    // M25 and M26 are coupled with M25 as the leader.
    // The motors cannot be set to always enabled, because they have brakes that
    // only activate when the motors are not moving. Due to the weight
    // of the frame, it appears that if the brake is not on, the motors
    // are moving constantly to keep the frame from falling. So essentially,
    // "is moving" is synonymous with "is enabled" for these motors which
    // results in the brake only applying if the motors are disabled. Setting M25
    // to only enable during motion, and M26 to NEVER means that
    // M25 will be enabled when commanded to move from EPICS but
    // for M26 the FB_MotionStage will not modify the bEnable boolean
    // in the state machine. Therefore, we can set the M26 bEnable
    // status based on the M25 bEnable status after the M25 FB_MotionStage
    // runs. But this also allows the brake to still activate when M26 is
    // not moving.
    Main.M25.nEnableMode := ENUM_StageEnableMode.NEVER ;
    // M26 bEnable is coupled to M25 bEnable below. Set M26 enable mode to NEVER
    // so that the function block does not try to set the bEnable bit unless
    // it detects an error. This allows the bEnable to be set outside of
    // the function block.
    Main.M26.nEnableMode := ENUM_StageEnableMode.NEVER ;

    Main.M27.nEnableMode := ENUM_StageEnableMode.DURING_MOTION ;
END_IF

stRenishawAbsEncMaster.Ref := 15370335;
stRenishawAbsEncSlave.Ref := 15347257;

// AutoCoupling
fbAutoCoupling(	nGantryTol 			:= 200000, // 50nm/count
                Master				:= Main.M25,
                MasterEnc			:= stRenishawAbsEncMaster,
                Slave				:= Main.M26,
                SlaveEnc			:= stRenishawAbsEncSlave,
                bExecuteCouple 		:= bExecuteCouple,
                bExecuteDecouple 	:= bExecuteDecouple,
);

// I don't think these 3 lines do anything but I am keeping for now.
// The FB_MotionStage overwrites the bAllEnable bit internally.
Main.M25.bAllEnable := Main.M25.bEnable AND GVL_EPS.bESTOP;
Main.M26.bAllEnable := Main.M26.bEnable AND GVL_EPS.bESTOP;
Main.M27.bAllEnable := Main.M27.bEnable AND GVL_EPS.bESTOP;

// Call Motion FB instance
IF NOT bDisableStateMachine THEN
    CASE nState OF
    -1:
        IF Main.M25.bExecute AND NOT (Main.M25.bError OR Main.M26.bError)  THEN
            Main.M25.bExecute := FALSE;
            Main.M25.bEnable := TRUE;
            nState := 0;
        ELSE
            Main.M25.bEnable := FALSE;
            Main.M25.bBrakeRelease := FALSE;
            Main.M26.bBrakeRelease := FALSE;
        END_IF
    0:
        tonDelay(IN:=TRUE, PT:=t#1s);
        IF tonDelay.Q THEN
            Main.M25.bBrakeRelease := TRUE;
            Main.M26.bBrakeRelease := TRUE;
            tonDelay(IN:=FALSE);
            nState := 1;
        ELSIF Main.M25.bError OR Main.M26.bError THEN
            nState := -1;
        END_IF
    1:
        tonDelay2(IN:=TRUE, PT:=t#1s);
        IF tonDelay2.Q THEN
            Main.M25.bExecute := TRUE;
            tonDelay2(IN:=FALSE);
            nState := 2;
        ELSIF Main.M25.bError OR Main.M26.bError THEN
            nState := -1;
        END_IF
    2:
        IF NOT Main.M25.bBusy AND NOT Main.M26.bBusy THEN
            nState := -1;
        END_IF
    100:
        nState := -1;
    END_CASE
END_IF

fbMotionYF1(stMotionStage:=Main.M25);

// Set the M26 bEnable equal to the M25 bEnable status to couple their enable bits together.
Main.M26.bEnable := Main.M25.bEnable;

fbMotionYF2(stMotionStage:=Main.M26);
fbMotionZF(stMotionStage:=Main.M27);

fbMeasureReferenceVelocity(
    stMotionStage:=Main.M25,
    nMicrostepsPerStep:=64,
    bBusy=>,
    fMeasuredReferenceVelocity=>
);

END_PROGRAM

// ---- Devices/FB_MeasureReferenceVelocity.TcPOU

FUNCTION_BLOCK FB_MeasureReferenceVelocity
VAR_IN_OUT
    stMotionStage: ST_MotionStage;
END_VAR
VAR_INPUT
    nMicrostepsPerStep: UINT := 64; // 64 for Beckhoff stepper drives EL7047, EL7037, EL7041, EL7031
END_VAR
VAR_OUTPUT
    bBusy: BOOL;
    fMeasuredReferenceVelocity: LREAL;
END_VAR
VAR
    nState: INT := -1;
    fbReadDriveAddress: MC_ReadDriveAddress;
    nMicrostepCounter AT %I*: UINT; // In microsteps (64 microsteps per step)
    bCounterOverflow AT %I*: BOOL;
    bCounterUnderflow AT %I*: BOOL;
    nMaxStepFrequencyBuffer: BYTE; // An enum corresponding to max step frequency
    fbReadCoEMaxStepFrequency: FB_ReadCoE;
    nMaxStepFrequency: UINT; // Fullsteps per Second
    fStartingInternalPosition: DINT;
    fEndingInternalPosition: DINT;
    fStartingEUPosition: LREAL;
    fEndingEUPosition: LREAL;
    fDeltaEUPosition: LREAL;
    fDeltaInternalPosition: LREAL;
    fDeltaSteps: LREAL;
    fEUPerStep: LREAL;

    rtOverflow: R_TRIG;
    rtUnderflow: R_TRIG;

    nDriveAddressReadState: INT := -1;
    bDriveAddressValid: BOOL;
END_VAR


CASE nDriveAddressReadState OF
-1:
    IF NOT bDriveAddressValid THEN
        nDriveAddressReadState := nDriveAddressReadState + 1;
        fbReadDriveAddress(
            Axis:=stMotionStage.Axis,
            Execute:=FALSE
        );
    END_IF
0: // Read drive address
    fbReadDriveAddress(
        Axis:=stMotionStage.Axis,
        Execute:=TRUE
    );
    IF NOT fbReadDriveAddress.Busy THEN
        nDriveAddressReadState := -1;
        bDriveAddressValid := TRUE;
    ELSIF fbReadDriveAddress.Error THEN
        nDriveAddressReadState := 100;
    END_IF
100:
    nDriveAddressReadState := -1;
END_CASE

CASE nState OF
-1:
    IF stMotionStage.bBusy AND bDriveAddressValid THEN
        nState := 0;
        fStartingInternalPosition := 0;
        fEndingInternalPosition := 0;
        rtOverflow(CLK:=bCounterOverflow);
        rtUnderflow(CLK:=bCounterUnderflow);
        fbReadCoEMaxStepFrequency(
            bExecute:=FALSE,
            pBuffer:=ADR(nMaxStepFrequencyBuffer)
        );
    ELSIF NOT bDriveAddressValid THEN
        nState := 100;
    END_IF
0: // A move has started so read the starting position information
    fbReadCoEMaxStepFrequency(
        bExecute:=TRUE,
        pBuffer:=ADR(nMaxStepFrequencyBuffer),
        sNetId:=stMotionStage.Axis.DriveAddress.NetID,
        nSlaveAddr:=stMotionStage.Axis.DriveAddress.SlaveAddress,
        nDesiredCoEIndex:=16#8012,
        nDesiredCoESubIndex:=5,
        nBufferLength:=1,
        bBusy=>,
        bError=>
    );
    IF fbReadCoEMaxStepFrequency.bBusy THEN
        nState := nState + 1;
    ELSIF fbReadCoEMaxStepFrequency.bError THEN
        nState := 100;
    END_IF
1:
    fbReadCoEMaxStepFrequency(
        bExecute:=TRUE,
        pBuffer:=ADR(nMaxStepFrequencyBuffer),
        sNetId:=stMotionStage.Axis.DriveAddress.NetID,
        nSlaveAddr:=stMotionStage.Axis.DriveAddress.SlaveAddress,
        nDesiredCoEIndex:=16#8012,
        nDesiredCoESubIndex:=5,
        nBufferLength:=1,
        bBusy=>,
        bError=>
    );
    IF NOT fbReadCoEMaxStepFrequency.bBusy THEN
        nState := nState + 1;
        fStartingEUPosition := stMotionStage.stAxisStatus.fActPosition;
        fStartingInternalPosition := nMicrostepCounter;

        CASE nMaxStepFrequencyBuffer OF
        0:
            nMaxStepFrequency := 1000;
        1:
            nMaxStepFrequency := 2000;
        2:
            nMaxStepFrequency := 4000;
        3:
            nMaxStepFrequency := 8000;
        4:
            nMaxStepFrequency := 16000;
        5:
            nMaxStepFrequency := 32000;
        END_CASE
    ELSIF fbReadCoEMaxStepFrequency.bError THEN
        nState := 100;
    END_IF
2: // Wait until the move ends and then read the last position information
    rtOverflow(CLK:=bCounterOverflow);
    rtUnderflow(CLK:=bCounterUnderflow);
    IF rtOverflow.Q THEN
        fEndingInternalPosition := fEndingInternalPosition + 65535;
    ELSIF rtUnderflow.Q THEN
        fEndingInternalPosition := fEndingInternalPosition - 65535;
    END_IF
    IF NOT stMotionStage.bBusy THEN
        nState := nState + 1;
        fEndingEUPosition := stMotionStage.stAxisStatus.fActPosition;
        fEndingInternalPosition := fEndingInternalPosition + nMicrostepCounter;
    END_IF
3: // Calculate the reference velocity from the measured move
    fDeltaEUPosition := fEndingEUPosition - fStartingEUPosition;
    fDeltaInternalPosition := fEndingInternalPosition - fStartingInternalPosition;
    fDeltaSteps := fDeltaInternalPosition / UINT_TO_LREAL(nMicrostepsPerStep);

    IF fDeltaSteps <> 0 THEN
        fEUPerStep := fDeltaEUPosition / fDeltaSteps;

        fMeasuredReferenceVelocity := UINT_TO_LREAL(nMaxStepFrequency) * fEUPerStep;
        nState := -1;
    ELSE
        nState := 100;
        fMeasuredReferenceVelocity := 0;
    END_IF
100: // Reserve for error handling
    nState := -1;
END_CASE

END_FUNCTION_BLOCK

// ---- Devices/FB_ReadCoE.TcPOU

FUNCTION_BLOCK FB_ReadCoE
VAR_INPUT
    bExecute: BOOL;
    pBuffer: PVOID; // ADR(buffer)
    sNetId: T_AmsNetId; // Have to be entered
    nSlaveAddr: UINT; // Have to be entered
    nDesiredCoEIndex: WORD; // Ex: CoE 16#9000 (9000:1)
    nDesiredCoESubIndex: Byte; // Ex: CoE 1 (9000:1)
    nBufferLength: UDINT; // number of bytes in the CoE to be read
END_VAR
VAR_OUTPUT
    bBusy: BOOL;
    bError: BOOL;
END_VAR
VAR
    fbCoERead: FB_EcCoESdoRead; // Function Block for reading from CoE
    nState: INT := -1; // RW-status
    rtExecute: R_TRIG;
END_VAR


CASE nState OF
-1:
    rtExecute(CLK:=bExecute);
    IF rtExecute.Q THEN
        nState := 0;
        bBusy := TRUE;
        bError := FALSE;
    ELSE
        bBusy := FALSE;
    END_IF
0:
   // Read entry
    fbCoERead(
       sNetId:= sNetId,
       nSlaveAddr:= nSlaveAddr,
       nSubIndex:= nDesiredCoeSubIndex,
       nIndex:= nDesiredCoEIndex,
       pDstBuf:= pBuffer,
       cbBufLen:= nBufferLength,
       bExecute:= FALSE,
       tTimeout:= T#1S
   );
   fbCoERead(
       sNetId:= sNetId,
       nSlaveAddr:= nSlaveAddr,
       nSubIndex:= nDesiredCoeSubIndex,
       nIndex:= nDesiredCoEIndex,
       pDstBuf:= pBuffer,
       cbBufLen:= nBufferLength,
       bExecute:= TRUE,
       tTimeout:= T#1S
   );
   nState := nState + 1; // Next state
1: // Execute CoE read until done
    fbCoERead(
       sNetId:= sNetId,
       nSlaveAddr:= nSlaveAddr,
       nSubIndex:= nDesiredCoeSubIndex,
       nIndex:= nDesiredCoEIndex,
       pDstBuf:= pBuffer,
       cbBufLen:= nBufferLength,
       bExecute:= TRUE,
       tTimeout:= T#1S
    );
    IF fbCoERead.bError THEN
      nState := 100;     // Error case
    ELSE
        IF NOT fbCoERead.bBusy THEN
            nState := -1;    // Done
            bBusy := FALSE;
        END_IF
    END_IF
100: // Error handling..
    nState := -1;
    bBusy := FALSE;
    bError := TRUE;
END_CASE

END_FUNCTION_BLOCK

// ---- Spectometer Arm POUs/PRG_DET_CHAMBER.TcPOU

PROGRAM PRG_DET_CHAMBER
VAR
    bInit: BOOL := TRUE;
    fbMotionXDC: FB_MotionStage;
    fbMotionRyDC: FB_MotionStage;
    fbMotionZDC: FB_MotionStage;
END_VAR


// Det. Chmber
IF bInit THEN
    bInit :=FALSE;
    Main.M22.bHardwareEnable:= TRUE;
    Main.M22.bPowerSelf:= TRUE;
    Main.M22.nBrakeMode:= ENUM_StageBrakeMode.NO_BRAKE;
    Main.M22.nEnableMode := ENUM_StageEnableMode.DURING_MOTION ;
    Main.M22.fVelocity := 0.1;

    Main.M23.bHardwareEnable:= TRUE;
    Main.M23.bPowerSelf:= TRUE;
    Main.M23.nBrakeMode:= ENUM_StageBrakeMode.NO_BRAKE;
    Main.M23.nEnableMode := ENUM_StageEnableMode.DURING_MOTION ;
    Main.M23.fVelocity := 0.1;

    Main.M24.bHardwareEnable:= TRUE;
    Main.M24.bPowerSelf:= TRUE;
    Main.M24.nBrakeMode:= ENUM_StageBrakeMode.NO_BRAKE;
    Main.M24.nEnableMode := ENUM_StageEnableMode.ALWAYS ; // This axis should always be enables due to belows
    Main.M24.fVelocity := 0.1;
END_IF;


fbMotionXDC(stMotionStage:= Main.M22);
fbMotionRyDC(stMotionStage:= Main.M23);
fbMotionZDC(stMotionStage:= Main.M24);

END_PROGRAM

// ---- Spectometer Arm POUs/PRG_DET_SLIT.TcPOU

PROGRAM PRG_DET_SLIT
VAR
    {attribute 'pytmc' := 'pv: QRIX:DETSL'}
    fbSlits_Det: FB_Slits;
    bExecuteMotion: BOOL := TRUE;
    bMoveOk: BOOL :=TRUE;
    bInit:BOOL:=TRUE;
END_VAR


// 4 jaws slit

IF bInit THEN
    bInit := FALSE;

    Main.M18.nBrakeMode := ENUM_StageBrakeMode.NO_BRAKE;
    Main.M18.bHardwareEnable := TRUE;
    Main.M18.bPowerSelf := TRUE;
    Main.M18.fVelocity := 0.1;

    Main.M19.nBrakeMode := ENUM_StageBrakeMode.NO_BRAKE;
    Main.M19.bHardwareEnable := TRUE;
    Main.M19.bPowerSelf := TRUE;
    Main.M19.fVelocity := 0.1;

    Main.M20.nBrakeMode := ENUM_StageBrakeMode.NO_BRAKE;
    Main.M20.bHardwareEnable := TRUE;
    Main.M20.bPowerSelf := TRUE;
    Main.M20.fVelocity := 0.1;

    Main.M21.nBrakeMode := ENUM_StageBrakeMode.NO_BRAKE;
    Main.M21.bHardwareEnable := TRUE;
    Main.M21.bPowerSelf := TRUE;
    Main.M21.fVelocity := 0.1;

    Main.M18.nEnableMode := ENUM_StageEnableMode.DURING_MOTION ;
    Main.M19.nEnableMode := ENUM_StageEnableMode.DURING_MOTION ;
    Main.M20.nEnableMode := ENUM_StageEnableMode.DURING_MOTION ;
    Main.M21.nEnableMode := ENUM_StageEnableMode.DURING_MOTION ;
END_IF
fbSlits_Det(	i_DevName:=					'DET_SLITS',
                stTopBlade:=				Main.M20,
                stBottomBlade:=				Main.M21,
                stLeftBlade:=				Main.M18,
                stRightBlade:=				Main.M19,
                io_fbFFHWO:=				GVL_PMPS.fbFastFaultOutput1,
                fbArbiter:=					GVL_PMPS.fbArbiter,
                bExecuteMotion:=			bExecuteMotion,
                bMoveOk:=					bMoveOk
);

END_PROGRAM

// ---- Devices/FB_Slits.TcPOU

FUNCTION_BLOCK FB_Slits
VAR_IN_OUT
    stTopBlade: ST_MotionStage;
    stBottomBlade: ST_MotionStage;
    stLeftBlade: ST_MotionStage; // Left Slit from upstream view
    stRightBlade: ST_MotionStage; // Right Slit from upstream view
    bExecuteMotion:BOOL ;
    io_fbFFHWO    :    FB_HardwareFFOutput;
    fbArbiter: FB_Arbiter();
END_VAR

VAR_INPUT

    {attribute 'pytmc' := '
    pv: PMPS_OK;
    io: i;
    field: ZNAM False
    field: ONAM True
    '}
    bMoveOk:BOOL;

    (*Offsets*)
    {attribute 'pytmc' := '
    pv: Offset_Top;
    io: io;
    '}
    rEncoderOffsetTop: REAL;
    {attribute 'pytmc' := '
    pv: ZeroOffset_Bottom;
    io: io;
    '}
    rEncoderOffsetBottom: REAL;

    {attribute 'pytmc' := 'pv: ZeroOffset_Left; io: io;'}
    rEncoderOffsetLeft: REAL;

    {attribute 'pytmc' := '
    pv: ZeroOffset_Right;
    io: io;
    '}
    rEncoderOffsetRight: REAL;
    i_DevName : STRING; //device name for FFO and PMPS diagnostics
    {attribute 'pytmc' := '
    pv: Home;
    io: i;
    field: ZNAM False
    field: ONAM True
    '}
    bHome:BOOL:=FALSE;
END_VAR

VAR
    fbTopBlade: FB_MotionStage;
    fbBottomBlade: FB_MotionStage;
    fbLeftBlade: FB_MotionStage;
    fbRightBlade: FB_MotionStage;
    fPosTopBlade: LREAL;
    fPosBottomBlade: LREAL;
    fPosLeftBlade: LREAL;
    fPosRightBlade: LREAL;

    bCollisionLimitationVert: BOOL;
    bCollisionLimitationHorz: BOOL;

    (*Motion Parameters*)
    fSmallDelta: LREAL := 0.01;
    fBigDelta: LREAL := 20;
    fMaxVelocity: LREAL := 0.5;
    fHighAccel: LREAL := 0.8;
    fLowAccel: LREAL := 0.1;

    stTop: ST_PositionState;
    stBOTTOM: ST_PositionState;
    stLeft: ST_PositionState;
    stRight: ST_PositionState;

    {attribute 'pytmc' := 'pv: TOP'}
    fbTop: FB_StatePTPMove;
    {attribute 'pytmc' := 'pv: BOTTOM'}
    fbBottom: FB_StatePTPMove;
    {attribute 'pytmc' := 'pv: LEFT'}
    fbLeft: FB_StatePTPMove;
    {attribute 'pytmc' := 'pv: RIGHT'}
    fbRight: FB_StatePTPMove;

    (*EPICS pvs*)
    {attribute 'pytmc' := '
    pv: XWID_REQ;
    io: io;
    '}
    rReqApertureSizeX : REAL;
    {attribute 'pytmc' := '
    pv: YWID_REQ;
    io: io;
    '}
    rReqApertureSizeY : REAL;
    {attribute 'pytmc' := '
    pv: XCEN_REQ;
    io: io;
    '}
    rReqCenterX: REAL;
    {attribute 'pytmc' := '
    pv: YCEN_REQ;
    io: io;
    '}
    rReqCenterY: REAL;

    {attribute 'pytmc' := '
    pv: ACTUAL_XWIDTH;
    io: io;
    '}
    rActApertureSizeX : REAL;

    {attribute 'pytmc' := '
    pv: ACTUAL_YWIDTH;
    io: io;
    '}
    rActApertureSizeY : REAL;
    {attribute 'pytmc' := '
    pv: ACTUAL_XCENTER;
    io: io;
    '}
    rActCenterX: REAL;
    {attribute 'pytmc' := '
    pv: ACTUAL_YCENTER;
    io: io;
    '}
    rActCenterY: REAL;

    {attribute 'pytmc' := '
    pv: XCEN_SETZERO;
    io: io;
    '}
    rSetCenterX: BOOL;
    {attribute 'pytmc' := '
    pv: YCEN_SETZERO;
    io: io;
    '}
    rSetCenterY: BOOL;


    {attribute 'pytmc' := '
    pv: OPEN;
    io: io;
    field: ZNAM False
    field: ONAM True
    '}
    bOpen: BOOL;

    {attribute 'pytmc' := '
    pv: CLOSE;
    io: io;
    field: ZNAM False
    field: ONAM True
    '}
    bClose: BOOL;

    {attribute 'pytmc' := '
    pv: BLOCK;
    io: io;
    field: ZNAM False
    field: ONAM True
    '}
    bBlock: BOOL;


     {attribute 'pytmc' := '
    pv: HOME_READY;
    io: i;
    field: ZNAM False
    field: ONAM True
    '}
    bHomeReady:BOOL:=FALSE;


    //Local variables
    bInit: BOOL :=true;
    rTrig_Block: R_TRIG;
    rTrig_Open: R_TRIG;
    rTrig_Close: R_TRIG;

    //old values
    rOldReqApertureSizeX : REAL;
    rOldReqApertureSizeY : REAL;
    rOldReqCenterX: REAL;
    rOldReqCenterY: REAL;

    bExecuteMotionX: BOOL;
    bExecuteMotionY: BOOL;


    fPosBlock: LREAL;
    fPosClose: LREAL;
    fPosOpen: LREAL;

    stSetPositionOptions:ST_SetPositionOptions;
    fbSetPosition_TOP: MC_SetPosition;
    fbSetPosition_Bottom: MC_SetPosition;
    fbSetPosition_Left: MC_SetPosition;
    fbSetPosition_Right: MC_SetPosition;

    // For logging
    fbLogger : FB_LogMessage := (eSubsystem:=E_SubSystem.MOTION);
    tErrorPresent : R_TRIG;
    tAction : R_TRIG;
    tOverrideActivated : R_TRIG;

    FFO    :    FB_FastFault :=(
        i_DevName := 'Slits',
        i_Desc := 'Fault occurs when center is greated than that requested',
        i_TypeCode := 16#1010);


    bTest: BOOL;

    AptArrayStatus AT %Q* : ST_PMPS_Aperture_IO;
    AptArrayReq AT %I* : ST_PMPS_Aperture_IO;

    fbPower: MC_Power;
END_VAR


// Initialize
ACT_init();
// Instantiate Function block for all the blades
ACT_Motion();
//SET and GET the requested and Actual values
ACT_CalculatePositions();

// Software Limits to protect blades
ACT_VirtualLimitSW();

ACTION ACT_BLOCK:

rTrig_Block (CLK:= bBlock);
rTrig_Open (CLK:= bOpen);
rTrig_Close (CLK:= bClose);

if (rTrig_Block.Q) THEN
    //BLOCK

    bBlock := false;
END_IF

if (rTrig_Open.Q) THEN


    bOpen := false;
END_IF

if (rTrig_Close.Q) THEN


    bClose := false;
END_IF
END_ACTION

ACTION ACT_CalculatePositions:

//check if requested center or gap has changed
//check that the requested values are within acceptable motion range
IF (rOldReqApertureSizeX <> rReqApertureSizeX) THEN
        rOldReqApertureSizeX := rReqApertureSizeX;
        bExecuteMotionX := TRUE;
        fbLogger(sMsg:='Requested new X gap.', eSevr:=TcEventSeverity.Verbose);
END_IF

IF (rOldReqCenterX <> rReqCenterX) THEN
    rOldReqCenterX := rReqCenterX;
    bExecuteMotionX := TRUE;
    fbLogger(sMsg:='Requested new X center', eSevr:=TcEventSeverity.Verbose);
   // ELSE
      //  rReqCenterX := rActCenterX;
END_IF

IF (rOldReqApertureSizeY <> rReqApertureSizeY) THEN
        rOldReqApertureSizeY := rReqApertureSizeY;
        bExecuteMotionY := TRUE;
        fbLogger(sMsg:='Requested new Y gap.', eSevr:=TcEventSeverity.Verbose);

END_IF

IF (rOldReqCenterY <> rReqCenterY) THEN
    rOldReqCenterY := rReqCenterY;
    bExecuteMotionY := TRUE;
    fbLogger(sMsg:='Requested new Y center.', eSevr:=TcEventSeverity.Verbose);
   // ELSE
      //  rReqCenterY := rActCenterY;
END_IF


//Calculate requested target positions from requested gap and center
fPosTopBlade := (rReqApertureSizeY/2) + (rReqCenterY + rEncoderOffsetTop) ;
fPosBottomBlade := (-1*rReqApertureSizeY/2) + (rReqCenterY+rEncoderOffsetBottom);

fPosLeftBlade := (rReqApertureSizeX/2) + (rReqCenterX + rEncoderOffsetLeft);
fPosRightBlade := (-1*rReqApertureSizeX/2) + (rReqCenterX + rEncoderOffsetRight);


//Calculate actual gap and center from actual stages positions
rActApertureSizeX := LREAL_TO_REAL((stLeftBlade.stAxisStatus.fActPosition - rEncoderOffsetLeft) - (stRightBlade.stAxisStatus.fActPosition- rEncoderOffsetRight));

rActApertureSizeY := LREAL_TO_REAL((stTopBlade.stAxisStatus.fActPosition - rEncoderOffsetTop) - (stBottomBlade.stAxisStatus.fActPosition - rEncoderOffsetBottom));

rActCenterX := LREAL_TO_REAL((((stLeftBlade.stAxisStatus.fActPosition - rEncoderOffsetLeft)  + (stRightBlade.stAxisStatus.fActPosition - rEncoderOffsetRight ))/2));

rActCenterY := LREAL_TO_REAL((((stTopBlade.stAxisStatus.fActPosition - rEncoderOffsetTop) + (stBottomBlade.stAxisStatus.fActPosition - rEncoderOffsetBottom))/2));


// Prevent collision
bCollisionLimitationHorz	:= (rActApertureSizeX > -0.1);
bCollisionLimitationVert	:= (rActApertureSizeY > -0.1);
END_ACTION

ACTION ACT_Init:

//  init the motion stages parameters
IF ( bInit) THEN
    stTopBlade.bHardwareEnable := TRUE;
    stBottomBlade.bHardwareEnable := TRUE;
    stLeftBlade.bHardwareEnable := TRUE;
    stRightBlade.bHardwareEnable := TRUE;
    stTopBlade.bPowerSelf :=FALSE;
    stBottomBlade.bPowerSelf :=FALSE;
    stLeftBlade.bPowerSelf :=FALSE;
    stRightBlade.bPowerSelf :=FALSE;
    stTopBlade.nBrakeMode := ENUM_StageBrakeMode.NO_BRAKE;
    stBottomBlade.nBrakeMode := ENUM_StageBrakeMode.NO_BRAKE;
    stLeftBlade.nBrakeMode := ENUM_StageBrakeMode.NO_BRAKE;
    stRightBlade.nBrakeMode := ENUM_StageBrakeMode.NO_BRAKE;
    FFO.i_DevName := i_DevName;
END_IF
END_ACTION

ACTION ACT_Motion:

// Instantiate Function block for all the blades
fbTopBlade(stMotionStage:=stTopBlade);
fbBottomBlade(stMotionStage:=stBottomBlade);
fbLeftBlade(stMotionStage:=stLeftBlade);
fbRightBlade(stMotionStage:=stRightBlade);



// PTP Motion for each blade
stTop.sName := 'Top';
stTop.fPosition := fPosTopBlade;
stTop.fDelta := fSmallDelta;
stTop.fVelocity := fMaxVelocity;
stTop.fAccel := fHighAccel;
stTop.fDecel := fHighAccel;

stBOTTOM.sName := 'Bottom';
stBOTTOM.fPosition := fPosBottomBlade;
stBOTTOM.fDelta := fSmallDelta;
stBOTTOM.fVelocity := fMaxVelocity;
stBOTTOM.fAccel := fHighAccel;
stBOTTOM.fDecel := fHighAccel;

stLeft.sName := 'Left';
stLeft.fPosition := fPosLeftBlade;
stLeft.fDelta := fSmallDelta;
stLeft.fVelocity := fMaxVelocity;
stLeft.fAccel := fHighAccel;
stLeft.fDecel := fHighAccel;

stRight.sName := 'Right';
stRight.fPosition := fPosRightBlade;
stRight.fDelta := fSmallDelta;
stRight.fVelocity := fMaxVelocity;
stRight.fAccel := fHighAccel;
stRight.fDecel := fHighAccel;

IF (bExecuteMotionY) THEN
    fbTop.bExecute := fbBottom.bExecute := bExecuteMotionY;
    bExecuteMotionY:= FALSE;
END_IF

IF (bExecuteMotionX) THEN
    fbLeft.bExecute := fbRight.bExecute := bExecuteMotionX;
    bExecuteMotionX:= FALSE;
END_IF


fbTop(
    stPositionState:=stTop,
    bMoveOk:=bMoveOk,
    stMotionStage:=stTopBlade);

fbBottom(
    stPositionState:=stBOTTOM,
    bMoveOk:=bMoveOk,
    stMotionStage:=stBottomBlade);

fbLeft(
    stPositionState:=stLeft,
    bMoveOk:=bMoveOk,
    stMotionStage:=stLeftBlade);

fbRight(
    stPositionState:=stRight,
    bMoveOk:=bMoveOk,
    stMotionStage:=stRightBlade);
END_ACTION

ACTION ACT_VirtualLimitSW:

// Force set to false
stLeftBlade.bPowerSelf := stRightBlade.bPowerSelf := stTopBlade.bPowerSelf := stBottomBlade.bPowerSelf := FALSE;

// Set SafetyReady flags manually
stTopBlade.bSafetyReady:= TRUE;
stBottomBlade.bSafetyReady:= TRUE;
stLeftBlade.bSafetyReady:= TRUE;
stRightBlade.bSafetyReady:= TRUE;


// Note: FB_MotionStage calls FB_SetEnables internally that overwrites .bAllForwardEnable/.bAllBackwardEnable flags

fbPower(
    Axis := stTopBlade.Axis,
    Enable := stTopBlade.bAllEnable,
    Enable_Positive := stTopBlade.bAllForwardEnable,
    Enable_Negative := stTopBlade.bAllBackwardEnable AND bCollisionLimitationVert,
    Override := 100.000
);
fbPower(
    Axis := stBottomBlade.Axis,
    Enable := stBottomBlade.bAllEnable,
    Enable_Positive := stBottomBlade.bAllForwardEnable AND bCollisionLimitationVert,
    Enable_Negative := stBottomBlade.bAllBackwardEnable,
    Override := 100.000
);
fbPower(
    Axis := stLeftBlade.Axis,
    Enable := stLeftBlade.bAllEnable,
    Enable_Positive := stLeftBlade.bAllForwardEnable,
    Enable_Negative := stLeftBlade.bAllBackwardEnable AND bCollisionLimitationHorz,
    Override := 100.000
);
fbPower(
    Axis := stRightBlade.Axis,
    Enable := stRightBlade.bAllEnable,
    Enable_Positive := stRightBlade.bAllForwardEnable AND bCollisionLimitationHorz,
    Enable_Negative := stRightBlade.bAllBackwardEnable,
    Override := 100.000
);
END_ACTION

END_FUNCTION_BLOCK

// ---- Spectometer Arm POUs/PRG_DET_FRAME.TcPOU

PROGRAM PRG_DET_FRAME
VAR
    bInit: BOOL := TRUE;
    {attribute 'pytmc' := '
        pv: QRIX:SA:bError
        io: i
    '}
    bError: BOOL := FALSE;
    {attribute 'pytmc' := '
        pv: QRIX:SA:bBusy
        io: i
    '}
    bBusy: BOOL;
    {attribute 'pytmc' := '
        pv: QRIX:SA:bMotorsBusy
        io: i
    '}
    bMotorsBusy: BOOL;
    {attribute 'pytmc' := 'pv: QRIX:SA:bResetError'}
    bResetError: BOOL := FALSE;
    {attribute 'pytmc' := 'pv: QRIX:SA:EnableJackOff'}
    bEnableJackOff: BOOL;
    {attribute 'pytmc' := 'pv: QRIX:SA:EnableLevitation'}
    bEnableLevitation: BOOL;
    {attribute 'pytmc' := 'pv: QRIX:SA:EnableLanding'}
    bEnableLanding: BOOL;
    {attribute 'pytmc' := 'pv: QRIX:DF:EnableAdjustingRoll'}
    bEnableAdjustingRoll: BOOL;
    {attribute 'pytmc' := 'pv: QRIX:DF:EnableAdjustingPitch'}
    bEnableAdjustingPitch: BOOL;
    {attribute 'pytmc' := 'pv: QRIX:DF:EnableAdjustingHeight'}
    bEnableAdjustingHeight: BOOL;

    tonWaitToStabilize: TON;

    tonSV2Open: TON;
    tonSV1Close: TON;

    tonDelayTrig: TON;

    iStepJackOff: INT := 1;
    iStepAdjustingRoll : INT := 1;
    iStepAdjustingPitch : INT := 1;
    iStepAdjustingHeight : INT := 1;

    trigDone: F_TRIG;

    fDistanceX: LREAL := 2.114; // in m
    fDistanceZ: LREAL := 2.142; // in m

    fPositionThreshold: LREAL := 0.02; // mm
    fPositionMaxDeviation: LREAL := 10.0; // mm
    fPitchThreshold: LREAL := 0.02; // mrad
    fRollThreshold: LREAL := 0.02; // mrad

    {attribute 'pytmc' := '
        pv: QRIX:SA:fRollTarget
        io: io
    '}
    fRollTarget : LREAL;

    {attribute 'pytmc' := 'pv: QRIX:F'}
    fbYDFMotion: FB_3AxesJack;

    fbReset_M15: MC_RESET;
    fbReset_M16: MC_RESET;
    fbReset_M17: MC_RESET;

    nActiveSequenceIterationCount: UINT := 1;
    nSequenceIterationCount: UINT := 3;

    // EPS settings to prevent jacks from moving too far out of range of each other.
    EPS_YDF1_Up   : FB_EPS;
    EPS_YDF1_Down : FB_EPS;
    EPS_YDF2_Up   : FB_EPS;
    EPS_YDF2_Down : FB_EPS;
    EPS_YDF3_Up   : FB_EPS;
    EPS_YDF3_Down : FB_EPS;

    {attribute 'pytmc' := '
        pv: QRIX:SA:rJackingSpeed
        io: io
    '}
    rJackingSpeed: LREAL := 0.05;
    {attribute 'pytmc' := '
        pv: QRIX:SA:rJackingAccel
        io: io
    '}
    rJackingAccel: LREAL := 0.005;

    {attribute 'pytmc' := '
        pv: QRIX:SA:bStopAxes
        io: io
    '}
    bStopAxes: BOOL;

    {attribute 'TcLinkTo' := 'TIIB[Rack#2D LinearGaugeAmp (SC-HG1-ETC)]^Process Data(In)  TxPDO-Map^Sensor Warning}
    bLinearGaugeWarning AT %I* : BOOL;
    {attribute 'TcLinkTo' := 'TIIB[Rack#2D LinearGaugeAmp (SC-HG1-ETC)]^Process Data(In)  TxPDO-Map^Sensor Error}
    bLinearGaugeError AT %I* : BOOL;

    {attribute 'TcLinkToOSO' := '<0,1,2>TINC^NC-Task 1 SAF^Axes^M15 - YDF1^Enc^Inputs^In^nState1'}
    bLinearGaugeYDF1Ready AT %Q* : BOOL;
    {attribute 'TcLinkToOSO' := '<0,1,2>TINC^NC-Task 1 SAF^Axes^M16 - YDF2^Enc^Inputs^In^nState1'}
    bLinearGaugeYDF2Ready AT %Q* : BOOL;
    {attribute 'TcLinkToOSO' := '<0,1,2>TINC^NC-Task 1 SAF^Axes^M17 - YDF3^Enc^Inputs^In^nState1'}
    bLinearGaugeYDF3Ready AT %Q* : BOOL;
END_VAR


IF bInit THEN
    bInit := FALSE;

    Main.M15.nBrakeMode := ENUM_StageBrakeMode.NO_BRAKE;
    Main.M15.bHardwareEnable := TRUE;
    Main.M15.bPowerSelf := TRUE;

    Main.M16.nBrakeMode := ENUM_StageBrakeMode.NO_BRAKE;
    Main.M16.bHardwareEnable := TRUE;
    Main.M16.bPowerSelf := TRUE;

    Main.M17.nBrakeMode := ENUM_StageBrakeMode.NO_BRAKE;
    Main.M17.bHardwareEnable := TRUE;
    Main.M17.bPowerSelf := TRUE;

    Main.M15.nEnableMode := ENUM_StageEnableMode.DURING_MOTION;
    Main.M16.nEnableMode := ENUM_StageEnableMode.DURING_MOTION;
    Main.M17.nEnableMode := ENUM_StageEnableMode.DURING_MOTION;
END_IF;

// FRAME JACKS EPS RESTRICTIONS
// YDF1 Disable movement in upward (positive/forward) direction.
EPS_YDF1_Up(eps:=Main.M15.stEPSForwardEnable);
EPS_YDF1_Up.setDescription('UPWARD MOVEMENT ALLOWED IF: YDF1 - YDF2 < 10mm AND YDF1 - YDF3 < 10mm |'); // SET DESCRIPTION FOR BYTE INDICATOR LABELS
// Prevent YDF1 from rising any more if it is more than fPositionMaxDeviation above YDF2
EPS_YDF1_Up.setBit(nBits:= 1, bValue:= Main.M15.stAxisStatus.fActPosition - Main.M16.stAxisStatus.fActPosition < fPositionMaxDeviation);
// Prevent YDF1 from rising any more if it is more than fPositionMaxDeviation above YDF3
EPS_YDF1_Up.setBit(nBits:= 0, bValue:= Main.M15.stAxisStatus.fActPosition - Main.M17.stAxisStatus.fActPosition < fPositionMaxDeviation);

// YDF1 Disable movement in downward (negative/downward) direction.
EPS_YDF1_Down(eps:=Main.M15.stEPSBackwardEnable);
EPS_YDF1_Down.setDescription('DOWNWARD MOVEMENT ALLOWED IF: YDF1 - YDF2 > -10mm AND YDF1 - YDF3 > -10mm |'); // SET DESCRIPTION FOR BYTE INDICATOR LABELS
// Prevent YDF1 from lowering any more if it is more than fPositionMaxDeviation below YDF2
EPS_YDF1_Down.setBit(nBits:= 1, bValue:= Main.M15.stAxisStatus.fActPosition - Main.M16.stAxisStatus.fActPosition > -fPositionMaxDeviation);
// Prevent YDF1 from lowering any more if it is more than fPositionMaxDeviation below YDF3
EPS_YDF1_Down.setBit(nBits:= 0, bValue:= Main.M15.stAxisStatus.fActPosition - Main.M17.stAxisStatus.fActPosition > -fPositionMaxDeviation);

// YDF2 Disable movement in upward (positive/forward) direction.
EPS_YDF2_Up(eps:=Main.M16.stEPSForwardEnable);
EPS_YDF2_Up.setDescription('UPWARD MOVEMENT ALLOWED IF:  YDF2 - YDF1 < 10mm AND YDF2 - YDF3 < 10mm |'); // SET DESCRIPTION FOR BYTE INDICATOR LABELS
// Prevent YDF2 from rising any more if it is more than fPositionMaxDeviation above YDF1
EPS_YDF2_Up.setBit(nBits:= 1, bValue:= Main.M16.stAxisStatus.fActPosition - Main.M15.stAxisStatus.fActPosition < fPositionMaxDeviation);
// Prevent YDF2 from rising any more if it is more than fPositionMaxDeviation above YDF3
EPS_YDF2_Up.setBit(nBits:= 0, bValue:= Main.M16.stAxisStatus.fActPosition - Main.M17.stAxisStatus.fActPosition < fPositionMaxDeviation);

// YDF2 Disable movement in downward (negative/downward) direction.
EPS_YDF2_Down(eps:=Main.M16.stEPSBackwardEnable);
EPS_YDF2_Down.setDescription('DOWNWARD MOVEMENT ALLOWED IF: YDF2 - YDF1 > -10mm AND YDF2 - YDF3 > -10mm |'); // SET DESCRIPTION FOR BYTE INDICATOR LABELS
// Prevent YDF2 from lowering any more if it is more than fPositionMaxDeviation below YDF1
EPS_YDF2_Down.setBit(nBits:= 1, bValue:= Main.M16.stAxisStatus.fActPosition - Main.M15.stAxisStatus.fActPosition > -fPositionMaxDeviation);
// Prevent YDF2 from lowering any more if it is more than fPositionMaxDeviation below YDF3
EPS_YDF2_Down.setBit(nBits:= 0, bValue:= Main.M16.stAxisStatus.fActPosition - Main.M17.stAxisStatus.fActPosition > -fPositionMaxDeviation);

// YDF3 Disable movement in upward (positive/forward) direction.
EPS_YDF3_Up(eps:=Main.M17.stEPSForwardEnable);
EPS_YDF3_Up.setDescription('UPWARD MOVEMENT ALLOWED IF: YDF3 - YDF2 < 10mm AND YDF3 - YDF1 < 10mm |'); // SET DESCRIPTION FOR BYTE INDICATOR LABELS
// Prevent YDF3 from rising any more if it is more than fPositionMaxDeviation above YDF2
EPS_YDF3_Up.setBit(nBits:= 1, bValue:= Main.M17.stAxisStatus.fActPosition - Main.M16.stAxisStatus.fActPosition < fPositionMaxDeviation);
// Prevent YDF3 from rising any more if it is more than fPositionMaxDeviation above YDF1
EPS_YDF3_Up.setBit(nBits:= 0, bValue:= Main.M17.stAxisStatus.fActPosition - Main.M15.stAxisStatus.fActPosition < fPositionMaxDeviation);

// YDF3 Disable movement in downward (negative/downward) direction.
EPS_YDF3_Down(eps:=Main.M17.stEPSBackwardEnable);
EPS_YDF3_Down.setDescription('DOWNWARD MOVEMENT ALLOWED IF: YDF3 - YDF2 > -10mm AND YDF3 - YDF1 > -10mm |'); // SET DESCRIPTION FOR BYTE INDICATOR LABELS
// Prevent YDF3 from lowering any more if it is more than fPositionMaxDeviation below YDF2
EPS_YDF3_Down.setBit(nBits:= 1, bValue:= Main.M17.stAxisStatus.fActPosition - Main.M16.stAxisStatus.fActPosition > -fPositionMaxDeviation);
// Prevent YDF3 from lowering any more if it is more than fPositionMaxDeviation below YDF1
EPS_YDF3_Down.setBit(nBits:= 0, bValue:= Main.M17.stAxisStatus.fActPosition - Main.M15.stAxisStatus.fActPosition > -fPositionMaxDeviation);

GVL_Sensor.bFloating := GVL_Sensor.stPS1.fValue > 0.3 AND GVL_Sensor.stPS2.fValue > 0.18 AND GVL_Sensor.stPS3.fValue > 0.15;

bMotorsBusy := Main.M15.bBusy OR Main.M16.bBusy OR Main.M17.bBusy;

IF Main.M15.bError OR Main.M16.bError OR Main.M17.bError THEN
    bError := TRUE;
    iStepJackOff := -1;
    iStepAdjustingRoll := -1;
    iStepAdjustingPitch := -1;
    iStepAdjustingHeight := -1;
    IF NOT Main.M15.bError THEN
        Main.M15.bReset := TRUE;
    END_IF;
    IF NOT Main.M16.bError THEN
        Main.M16.bReset := TRUE;
    END_IF;
    IF NOT Main.M17.bError THEN
        Main.M17.bReset := TRUE;
    END_IF;
END_IF

ACT_1_JACK_OFF();
ACT_2_Levitation();
ACT_3_Landing();
ACT_4_AdjustingRoll();
ACT_5_AdjustingPitch();
ACT_6_AdjustingHeight();
ACT_ResetError();

bLinearGaugeYDF1Ready := NOT bLinearGaugeError;
bLinearGaugeYDF2Ready := NOT bLinearGaugeError;
bLinearGaugeYDF3Ready := NOT bLinearGaugeError;

fbYDFMotion(
    bMoveOk			  := GVL_EPS.bESTOP,
    stJack1Axis		  := Main.M16,
    stJack2Axis		  := Main.M15,
    stJack3Axis		  := Main.M17,
    rDistanceX        := fDistanceX,
    rDistanceZ        := fDistanceZ,
    bJack3DoesPitch   :=  TRUE,
    rLimitPositionMax :=  21.5,
    rLimitPositionMin := -0.5,
    rLimitPitchMin    := -10,
    rLimitPitchMax    :=  10,
    rLimitRollMin     := -10,
    rLimitRollMax     :=  10,
    fMaxVelocity      :=  rJackingSpeed,
    fHighAccel        :=  rJackingAccel
);

IF bStopAxes THEN
    Main.M1.bExecute := FALSE;
    Main.M2.bExecute := FALSE;
    Main.M7.bExecute := FALSE;
    Main.M8.bExecute := FALSE;
    Main.M9.bExecute := FALSE;
    Main.M15.bExecute := FALSE;
    Main.M16.bExecute := FALSE;
    Main.M17.bExecute := FALSE;
    bStopAxes := FALSE;
END_IF

ACTION ACT_1_JACK_OFF:

CASE iStepJackOff OF
    1:
        IF bEnableJackOff AND NOT(bBusy AND bError) THEN
            iStepJackOff := 2;
            bDoneJackOff := FALSE;
            bBusy := TRUE;
            fbYDFMotion.bMoveToPosition := FALSE;
            fbYDFMotion.bMoveToPitch := FALSE;
            fbYDFMotion.bMoveToRoll := FALSE;
        ELSE
            bEnableJackOff := FALSE;
        END_IF;
    2:
        // Step2 check if we are already at position or if we are in an error position.
        IF abs(Main.M15.stAxisStatus.fActPosition) < fPositionThreshold AND
           abs(Main.M16.stAxisStatus.fActPosition) < fPositionThreshold AND
           abs(Main.M17.stAxisStatus.fActPosition) < fPositionThreshold THEN
            // We dont need to move any more....
            iStepJackOff := 4;
        ELSE
            iStepJackOff := 3;
        END_IF;
    3:
        // Step3 set target position
        fbYDFMotion.rReqPosition := 0.0;
        fbYDFMotion.bMoveToPosition := TRUE;
        fbYDFMotion.rReqRoll := 0.0;
        fbYDFMotion.bMoveToRoll := TRUE;
        fbYDFMotion.rReqPitch := 0.0;
        fbYDFMotion.bMoveToPitch := TRUE;

        iStepJackOff := 2;
    4:
        // End
        bEnableJackOff:= FALSE;
        bBusy := FALSE;
        iStepJackOff:=1;
        bDoneJackOff := TRUE;
        fbYDFMotion.bMoveToPosition := FALSE;
        fbYDFMotion.bMoveToPitch := FALSE;
        fbYDFMotion.bMoveToRoll := FALSE;
    -1:
        // Error
        bError:= TRUE;
        bEnableJackOff:= FALSE;
        bBusy := FALSE;
        iStepJackOff:=1;
        bDoneJackOff := FALSE;
        fbYDFMotion.bMoveToPosition := FALSE;
        fbYDFMotion.bMoveToPitch := FALSE;
        fbYDFMotion.bMoveToRoll := FALSE;

END_CASE;
END_ACTION

ACTION ACT_2_Levitation:

IF bEnableLevitation AND NOT (bBusy OR bError) THEN
    bBusy := TRUE;
    IF GVL_Sensor.stPS1.fValue > 0.15 AND GVL_Sensor.stPS2.fValue > 0.15 THEN
        GVL_EPS.bOpenSV1 := TRUE;
    END_IF;
    bDoneLevitation := FALSE;
END_IF;

// SV2 will open after 3 secounds from SV1 opened...
tonSV2Open(
    IN := bEnableLevitation AND GVL_EPS.bOpenSV1,
    PT := T#3s
);

IF tonSV2Open.Q THEN
    GVL_EPS.bOpenSV2 := TRUE;
    bEnableLevitation := FALSE;
    bDoneLevitation := TRUE;
    bBusy := FALSE;
END_IF;
END_ACTION

ACTION ACT_3_Landing:

IF bEnableLanding AND NOT (bBusy OR bError) THEN
    GVL_EPS.bOpenSV2 := FALSE;
    bBusy:= TRUE;
    bDoneLanding := FALSE;
END_IF;

tonSV1Close(
    IN := bEnableLanding AND NOT GVL_EPS.bOpenSV2,
    PT := T#3s
);

IF tonSV1Close.Q THEN
    GVL_EPS.bOpenSV1 := FALSE;
    bEnableLanding := FALSE;
    bBusy:= FALSE;
    bDoneLanding := TRUE;
END_IF;
END_ACTION

ACTION ACT_4_AdjustingRoll:

CASE iStepAdjustingRoll OF
    1:
        IF bEnableAdjustingRoll AND NOT(bBusy AND bError) THEN
            iStepAdjustingRoll := 2;
            bDoneAdjustingRoll := FALSE;
            bBusy := TRUE;
            fbYDFMotion.bMoveToRoll := FALSE;
            nActiveSequenceIterationCount := 0;
        ELSE
            bEnableAdjustingRoll := FALSE;
        END_IF;
    2:
        // Step3 set target roll
        IF abs(GVL_Sensor.stFrameR.fValue - fRollTarget) > fRollThreshold THEN
            fbYDFMotion.bMoveToRoll := TRUE;
            iStepAdjustingRoll := 3;
            fbYDFMotion.rReqRoll := fbYDFMotion.rActRoll - (GVL_Sensor.stFrameR.fValue - fRollTarget) * 0.5;
        ELSE
            // Already at goal.
            iStepAdjustingRoll := 4;
        END_IF;
    3:
        // Wait until Done. and wait tilt sensor stabilization.
        tonWaitToStabilize(IN:=NOT bMotorsBusy, PT:=T#5s);
        IF tonWaitToStabilize.Q THEN
            iStepAdjustingRoll := 4;
            tonWaitToStabilize(IN:=FALSE);
        END_IF;
    4:
        IF nActiveSequenceIterationCount > nSequenceIterationCount THEN
            // Exceeded maximum allowable number of iterations. Something is wrong.
            iStepAdjustingRoll := -1;
        ELSIF abs(GVL_Sensor.stFrameR.fValue - fRollTarget) > fRollThreshold THEN
            // Iteration
            iStepAdjustingRoll := 2;
            fbYDFMotion.bMoveToRoll := FALSE;
            nActiveSequenceIterationCount := nActiveSequenceIterationCount + 1;
        ELSE
            // End
            bEnableAdjustingRoll:= FALSE;
            bBusy := FALSE;
            iStepAdjustingRoll:=1;
            bDoneAdjustingRoll := TRUE;
            fbYDFMotion.bMoveToRoll := FALSE;
        END_IF;
    -1:
        // Error
        bError:= TRUE;
        bBusy := FALSE;
        bEnableAdjustingRoll:= FALSE;
        iStepAdjustingRoll:=1;
        bDoneAdjustingRoll := FALSE;
        fbYDFMotion.bMoveToRoll := FALSE;
END_CASE;
END_ACTION

ACTION ACT_5_AdjustingPitch:

CASE iStepAdjustingPitch OF
    1:
        IF bEnableAdjustingPitch AND NOT(bBusy AND bError) THEN
            iStepAdjustingPitch := 2;
            bDoneAdjustingPitch := FALSE;
            bBusy := TRUE;
            fbYDFMotion.bMoveToPitch := FALSE;
            nActiveSequenceIterationCount := 0;
        ELSE
            bEnableAdjustingPitch := FALSE;
        END_IF;
    2:
        // Step2 set target pitch
        IF abs(GVL_Sensor.stFrameP.fValue) > fPitchThreshold THEN
            fbYDFMotion.bMoveToPitch := TRUE;
            iStepAdjustingPitch := 3;
            fbYDFMotion.rReqPitch := fbYDFMotion.rActPitch - GVL_Sensor.stFrameP.fValue * 0.5;
        ELSE
            // Already at goal.
            iStepAdjustingPitch := 4;
        END_IF;
    3:
        // Wait until Done. and wait tilt sensor stabilization.
        tonWaitToStabilize(IN:=NOT bMotorsBusy, PT:=T#5s);
        IF tonWaitToStabilize.Q THEN
            iStepAdjustingPitch := 4;
            tonWaitToStabilize(IN:=FALSE);
        END_IF;
    4:
        IF nActiveSequenceIterationCount > nSequenceIterationCount THEN
            // Exceeded maximum allowable number of iterations. Something is wrong.
            iStepAdjustingPitch := -1;
        ELSIF abs(GVL_Sensor.stFrameP.fValue) > fPitchThreshold THEN
            // Iteration
            iStepAdjustingPitch := 2;
            fbYDFMotion.bMoveToPitch := FALSE;
            nActiveSequenceIterationCount := nActiveSequenceIterationCount + 1;
        ELSE
            // End
            bEnableAdjustingPitch:= FALSE;
            bBusy := FALSE;
            iStepAdjustingPitch:=1;
            bDoneAdjustingPitch := TRUE;
            fbYDFMotion.bMoveToPitch := FALSE;
        END_IF;
    -1:
        // Error
        bError:= TRUE;
        bBusy := FALSE;
        bEnableAdjustingPitch:= FALSE;
        iStepAdjustingPitch:=1;
        bDoneAdjustingPitch := FALSE;
        fbYDFMotion.bMoveToPitch := FALSE;
END_CASE;
END_ACTION

ACTION ACT_6_AdjustingHeight:

CASE iStepAdjustingHeight OF
    1:
        IF bEnableAdjustingHeight AND NOT(bBusy AND bError) THEN
            iStepAdjustingHeight := 2;
            bDoneAdjustingHeight := FALSE;
            bBusy := TRUE;
            fbYDFMotion.bMoveToPosition := FALSE;
            nActiveSequenceIterationCount := 0;
        ELSE
            bEnableAdjustingHeight := FALSE;
        END_IF;
    2:
        // Step2 set target position
        IF abs(GVL_Sensor.stHDF.fValue) > fPositionThreshold THEN
            fbYDFMotion.bMoveToPosition := TRUE;
            iStepAdjustingHeight := 3;
            fbYDFMotion.rReqPosition := fbYDFMotion.rActPosition - GVL_Sensor.stHDF.fValue;
        ELSE
            // Already at goal.
            iStepAdjustingHeight := 4;
        END_IF;
    3:
        // Wait until Done. and wait tilt sensor stabilization.
        tonWaitToStabilize(IN:=NOT bMotorsBusy, PT:=T#5s);
        IF tonWaitToStabilize.Q THEN
            iStepAdjustingHeight := 4;
            tonWaitToStabilize(IN:=FALSE);
        END_IF;
    4:
        IF nActiveSequenceIterationCount > nSequenceIterationCount THEN
            // Exceeded maximum allowable number of iterations. Something is wrong.
            iStepAdjustingHeight := -1;
        ELSIF abs(GVL_Sensor.stHDF.fValue) > fPositionThreshold THEN
            // Iteration
            iStepAdjustingHeight := 2;
            fbYDFMotion.bMoveToPosition := FALSE;
            nActiveSequenceIterationCount := nActiveSequenceIterationCount + 1;
        ELSE
            // End
            bEnableAdjustingHeight:= FALSE;
            bBusy := FALSE;
            iStepAdjustingHeight:=1;
            bDoneAdjustingHeight := TRUE;
            fbYDFMotion.bMoveToPosition := FALSE;
        END_IF;
    -1:
        // Error
        bError:= TRUE;
        bBusy := FALSE;
        bEnableAdjustingHeight:= FALSE;
        iStepAdjustingHeight:=1;
        bDoneAdjustingHeight := FALSE;
END_CASE;
END_ACTION

ACTION ACT_ResetError:

IF bResetError THEN
    bResetError := FALSE;
    bError:= FALSE;
    bBusy:=FALSE;
    bEnableJackOff := FALSE;
    bEnableLevitation := FALSE;
    bEnableLanding := FALSE;
    bEnableAdjustingRoll := FALSE;
    bEnableAdjustingPitch := FALSE;
    bEnableAdjustingHeight := FALSE;

    Main.M2.bReset := TRUE;
    Main.M2.bError := FALSE;

    (*Reset*)
    fbReset_M15(
        Execute:=Main.M15.Axis.Status.Error,
        Axis:=Main.M15.Axis,
        Done=> ,
        Busy=> ,
        Error=> ,
        ErrorID=> );
    fbReset_M16(
        Execute:=Main.M16.Axis.Status.Error,
        Axis:=Main.M16.Axis,
        Done=> ,
        Busy=> ,
        Error=> ,
        ErrorID=> );
    fbReset_M17(
        Execute:=Main.M17.Axis.Status.Error,
        Axis:=Main.M17.Axis,
        Done=> ,
        Busy=> ,
        Error=> ,
        ErrorID=> );

    iStepJackOff := 1;
    iStepAdjustingRoll := 1;
    iStepAdjustingPitch := 1;
    iStepAdjustingHeight := 1;

    fbYDFMotion.bMoveToPosition := FALSE;
    fbYDFMotion.bMoveToPitch := FALSE;
    fbYDFMotion.bMoveToRoll := FALSE;
    fbYDFMotion.rReqPosition := fbYDFMotion.rActPosition;
    fbYDFMotion.rReqPitch := fbYDFMotion.rActPitch;
    fbYDFMotion.rReqRoll := fbYDFMotion.rActRoll;

    bStopAxes := TRUE;
END_IF;
END_ACTION

END_PROGRAM

// ---- Devices/FB_3AxesJack.TcPOU

FUNCTION_BLOCK FB_3AxesJack
VAR_IN_OUT
    // Jack 1 is the axis that, when higher than Jack 2, creates a negative pitch/roll
    stJack1Axis: ST_MotionStage;
    // Jack 2 is the axis that, when higher than Jack1, creates a positive pitch/roll
    stJack2Axis: ST_MotionStage;
    // Jack 3 must be used as the jack that only contributes to Roll OR only contributes to Pitch
    // Assign your axes such that this jack is the jack that can only do roll OR pitch.
    // Jack 3 is assumed on the positive side of the pitch/roll, so to reverse the sign simply
    // supply a negative rDistanceX or rDistanceY, the choice of which is negative depends on
    // whether JAck3 is an axis that does only roll or only pitch.
    stJack3Axis: ST_MotionStage;
END_VAR
VAR_INPUT

    {attribute 'pytmc' := '
        pv: bMoveToPosition;
        io: i;
    '}
    bMoveToPosition: BOOL;
    {attribute 'pytmc' := '
        pv: bMoveToPitch;
        io: i;
    '}
    bMoveToPitch: BOOL;
    {attribute 'pytmc' := '
        pv: bMoveToRoll;
        io: i;
    '}
    bMoveToRoll: BOOL;

    {attribute 'pytmc' := '
    pv: PMPS_OK;
    io: i;
    field: ZNAM False
    field: ONAM True
    '}
    bMoveOk:BOOL;

    // Desired height, pitch, and roll
    {attribute 'pytmc' := '
    pv: Y_REQ;
    io: io;
    '}
    rReqPosition : REAL;

    {attribute 'pytmc' := '
    pv: PITCH_REQ;
    io: io;
    '}
    rReqPitch : REAL;

    {attribute 'pytmc' := '
    pv: ROLL_REQ;
    io: io;
    '}
    rReqRoll : REAL;

    (*Offsets*)
    {attribute 'pytmc' := '
    pv: ZeroOffset_Jack1;
    io: io;
    '}
    rEncoderOffsetJack1: REAL;

    {attribute 'pytmc' := '
    pv: ZeroOffset_Jack2;
    io: io;
    '}
    rEncoderOffsetJack2: REAL;

    {attribute 'pytmc' := '
    pv: ZeroOffset_Jack3;
    io: io;
    '}
    rEncoderOffsetJack3: REAL;

    // The distance along the pitch axis between the two sides of jacks.
    rDistanceX: REAL := 0.24;
    // The distance along the roll axis between the two sides of jacks.
    rDistanceZ: REAL := 0.88;
    bJack3DoesPitch: BOOL;

    rLimitPositionMax: REAL := 8;
    rLimitPositionMin: REAL := -8;
    rLimitPitchMin: REAL := -18;
    rLimitPitchMax: REAL :=  18;
    rLimitRollMin: REAL  := -18;
    rLimitRollMax: REAL  :=  18;

    (*Motion Parameters*)
    fSmallDelta: LREAL := 0.01;
    fBigDelta: LREAL := 10;
    fMaxVelocity: LREAL := 0.1;
    fHighAccel: LREAL := 0.8;
    fLowAccel: LREAL := 0.1;

     {attribute 'pytmc' := '
    pv: Home;
    io: i;
    field: ZNAM False
    field: ONAM True
    '}
    bHome:BOOL:=FALSE;
END_VAR

VAR
    fbJack1Stage: FB_MotionStage;
    fbJack2Stage: FB_MotionStage;
    fbJack3Stage: FB_MotionStage;
    fPosJack1Stage: LREAL;
    fPosJack2Stage: LREAL;
    fPosJack3Stage: LREAL;

    stJack1: ST_PositionState;
    stJack2: ST_PositionState;
    stJack3: ST_PositionState;

    {attribute 'pytmc' := 'pv: JACK1'}
    fbJack1: FB_StatePTPMove;
    {attribute 'pytmc' := 'pv: JACK2'}
    fbJack2: FB_StatePTPMove;
    {attribute 'pytmc' := 'pv: JACK3'}
    fbJack3: FB_StatePTPMove;

    //old values
    rOldReqPosition : REAL;
    rOldReqPitch: REAL;
    rOldReqRoll: REAL;

    (*EPICS pvs*)
    {attribute 'pytmc' := '
    pv: Y;
    io: i;
    '}
    rActPosition : REAL;

    {attribute 'pytmc' := '
    pv: PITCH;
    io: i;
    '}
    rActPitch : REAL;

    {attribute 'pytmc' := '
    pv: ROLL;
    io: i;
    '}
    rActRoll : REAL;


    {attribute 'pytmc' := '
    pv: HOME_READY;
    io: i;
    field: ZNAM False
    field: ONAM True
    '}
    bHomeReady:BOOL:=FALSE;


    //Local variables
    bInit: BOOL :=true;

    bExecuteMotionX: BOOL;

    fPosBlock: LREAL;
    fPosClose: LREAL;
    fPosOpen: LREAL;

    stSetPositionOptions: ST_SetPositionOptions;
    fbSetPosition_Pos: MC_SetPosition;
    fbSetPosition_Angle: MC_SetPosition;

    // For logging
    fbLogger : FB_LogMessage := (eSubsystem:=E_SubSystem.MOTION);
    tErrorPresent : R_TRIG;
    tAction : R_TRIG;
    tOverrideActivated : R_TRIG;

    bTest: BOOL;

    fbPower: MC_POWER;

    y1: LREAL;
    y2: LREAL;
    y3: LREAL;
    y12Ave: LREAL;
    y12Diff: LREAL;
END_VAR


// Instantiate Function block for all the blades
ACT_Motion();

//SET and GET the requested and Actual values
ACT_CalculatePositions();

// Software Limits to protect blades
ACT_VirtualLimitSW();

ACTION ACT_CalculatePositions:

//check if requested center or gap has changed
//check that the requested values are within acceptable motion range
IF abs(rReqPosition - rOldReqPosition) > 0.01 OR bMoveToPosition THEN
        rOldReqPosition := rReqPosition;
        bExecuteMotionX := TRUE;
        fbLogger(sMsg:='Requested new Position.', eSevr:=TcEventSeverity.Verbose);
ELSE
    rReqPosition := rActPosition;
    rOldReqPosition := rReqPosition;
END_IF

IF abs(rReqPitch - rOldReqPitch) > 0.01 OR bMoveToPitch THEN
    rOldReqPitch := rReqPitch;
    bExecuteMotionX := TRUE;
    fbLogger(sMsg:='Requested new Pitch', eSevr:=TcEventSeverity.Verbose);
ELSE
    rReqPitch := rActPitch;
    rOldReqPitch := rReqPitch;
END_IF

IF abs(rReqRoll - rOldReqRoll) > 0.01 OR bMoveToRoll THEN
    rOldReqRoll := rReqRoll;
    bExecuteMotionX := TRUE;
    fbLogger(sMsg:='Requested new Roll', eSevr:=TcEventSeverity.Verbose);
ELSE
    rReqRoll := rActRoll;
    rOldReqRoll := rReqRoll;
END_IF

//Calculate requested target positions from requested roll, pitch, and midpoint height.
IF bJack3DoesPitch THEN
    fPosJack1Stage := rReqPosition - rDistanceX / 2.0 * rReqRoll - rDistanceZ / 2.0 * rReqPitch + rEncoderOffsetJack1;
    fPosJack2Stage := rReqPosition + rDistanceX / 2.0 * rReqRoll - rDistanceZ / 2.0 * rReqPitch + rEncoderOffsetJack2;
    fPosJack3Stage := rReqPosition + rDistanceZ / 2.0 * rReqPitch + rEncoderOffsetJack3;
ELSE
    fPosJack1Stage := rReqPosition - rDistanceX / 2.0 * rReqRoll - rDistanceZ / 2.0 * rReqPitch + rEncoderOffsetJack1;
    fPosJack2Stage := rReqPosition - rDistanceX / 2.0 * rReqRoll + rDistanceZ / 2.0 * rReqPitch + rEncoderOffsetJack2;
    fPosJack3Stage := rReqPosition + rDistanceX / 2.0 * rReqRoll + rEncoderOffsetJack3;
END_IF;

//Calculate actual gap and center from actual stages positions
y1 := stJack1Axis.stAxisStatus.fActPosition;
y2 := stJack2Axis.stAxisStatus.fActPosition;
y3 := stJack3Axis.stAxisStatus.fActPosition;
y12Ave := (y1 + y2) / 2.0;
y12Diff := y2 - y1;

// Compute the actual height of the midpoint of the three jacks.
rActPosition := (y12Ave + y3) / 2;

// Compute the roll and pitch based on the the relative position of the three jacks.
IF bJack3DoesPitch THEN
    rActPitch := (y3 - y12Ave) / rDistanceZ;
    rActRoll  := y12Diff / rDistanceX;
ELSE
    rActRoll := (y3 - y12Ave) / rDistanceX;
    rActPitch  := y12Diff / rDistanceZ;
END_IF;
END_ACTION

ACTION ACT_Motion:

// Instantiate Function block for all the blades
fbJack1Stage(stMotionStage:=stJack1Axis);
fbJack2Stage(stMotionStage:=stJack2Axis);
fbJack3Stage(stMotionStage:=stJack3Axis);

// PTP Motion for each blade
stJack1.sName := 'Jack1';
stJack1.fPosition := fPosJack1Stage;
stJack1.fDelta := fSmallDelta;
stJack1.fVelocity := fMaxVelocity;
stJack1.fAccel := fHighAccel;
stJack1.fDecel := fHighAccel;

stJack2.sName := 'Jack2';
stJack2.fPosition := fPosJack2Stage;
stJack2.fDelta := fSmallDelta;
stJack2.fVelocity := fMaxVelocity;
stJack2.fAccel := fHighAccel;
stJack2.fDecel := fHighAccel;

stJack3.sName := 'Jack3';
stJack3.fPosition := fPosJack3Stage;
stJack3.fDelta := fSmallDelta;
stJack3.fVelocity := fMaxVelocity;
stJack3.fAccel := fHighAccel;
stJack3.fDecel := fHighAccel;

IF (bExecuteMotionX) THEN
    fbJack1.bExecute := fbJack2.bExecute := fbJack3.bExecute := bExecuteMotionX;
    bExecuteMotionX:= FALSE;
END_IF

fbJack1(
    stPositionState:=stJack1,
    bMoveOk:=bMoveOk,
    stMotionStage:=stJack1Axis);

fbJack2(
    stPositionState:=stJack2,
    bMoveOk:=bMoveOk,
    stMotionStage:=stJack2Axis);

fbJack3(
    stPositionState:=stJack3,
    bMoveOk:=bMoveOk,
    stMotionStage:=stJack3Axis);
END_ACTION

ACTION ACT_VirtualLimitSW:

// Set SafetyReady flags manually
stJack1Axis.bSafetyReady:= TRUE;
stJack2Axis.bSafetyReady:= TRUE;
stJack3Axis.bSafetyReady:= TRUE;

// Note: FB_MotionStage calls FB_SetEnables internally that overwrites .bAllForwardEnable/.bAllBackwardEnable flags
fbPower(
    Axis := stJack1Axis.Axis,
    Enable := stJack1Axis.bAllEnable,
    Enable_Positive := stJack1Axis.bAllForwardEnable  AND rActPosition <= rLimitPositionMax AND rActPitch <= rLimitPitchMax,
    Enable_Negative := stJack1Axis.bAllBackwardEnable AND rActPosition >= rLimitPositionMin AND rActPitch >= rLimitPitchMin,
    Override := 100.000
);
fbPower(
    Axis := stJack2Axis.Axis,
    Enable := stJack2Axis.bAllEnable,
    Enable_Positive := stJack2Axis.bAllForwardEnable  AND rActPosition <= rLimitPositionMax AND rActRoll <= rLimitRollMax,
    Enable_Negative := stJack2Axis.bAllBackwardEnable AND rActPosition >= rLimitPositionMin AND rActRoll >= rLimitRollMin,
    Override := 100.000
);
fbPower(
    Axis := stJack3Axis.Axis,
    Enable := stJack3Axis.bAllEnable,
    Enable_Positive := stJack3Axis.bAllForwardEnable  AND rActPosition <= rLimitPositionMax AND rActPitch >= rLimitPitchMin,
    Enable_Negative := stJack3Axis.bAllBackwardEnable AND rActPosition >= rLimitPositionMin AND rActPitch <= rLimitPitchMax,
    Override := 100.000
);
END_ACTION

END_FUNCTION_BLOCK

// ---- Spectometer Arm POUs/PRG_OPT_SLITS.TcPOU

PROGRAM PRG_OPT_SLITS
VAR
    {attribute 'pytmc' := 'pv: QRIX:OPTSL'}
    fbSlits_Opt: FB_Slits;
    bExecuteMotion: BOOL := TRUE;
    bMoveOk: BOOL :=TRUE;
    bInit:BOOl:=TRUE;
END_VAR


// 4 jaws slit



IF bInit THEN
    bInit := FALSE;

    Main.M3.nBrakeMode := ENUM_StageBrakeMode.NO_BRAKE;
    Main.M3.bHardwareEnable := TRUE;
    Main.M3.bPowerSelf := TRUE;
    Main.M3.fVelocity := 0.1;

    Main.M4.nBrakeMode := ENUM_StageBrakeMode.NO_BRAKE;
    Main.M4.bHardwareEnable := TRUE;
    Main.M4.bPowerSelf := TRUE;
    Main.M4.fVelocity := 0.1;

    Main.M5.nBrakeMode := ENUM_StageBrakeMode.NO_BRAKE;
    Main.M5.bHardwareEnable := TRUE;
    Main.M5.bPowerSelf := TRUE;
    Main.M5.fVelocity := 0.1;

    Main.M6.nBrakeMode := ENUM_StageBrakeMode.NO_BRAKE;
    Main.M6.bHardwareEnable := TRUE;
    Main.M6.bPowerSelf := TRUE;
    Main.M6.fVelocity := 0.1;


    //
    Main.M3.nEnableMode := ENUM_StageEnableMode.DURING_MOTION ;
    Main.M4.nEnableMode := ENUM_StageEnableMode.DURING_MOTION ;
    Main.M5.nEnableMode := ENUM_StageEnableMode.DURING_MOTION ;
    Main.M6.nEnableMode := ENUM_StageEnableMode.DURING_MOTION ;
END_IF



fbSlits_Opt(	i_DevName:=					'OPT_SLITS',
                stTopBlade:=				Main.M5,
                stBottomBlade:=				Main.M6,
                stLeftBlade:=				Main.M3,
                stRightBlade:=				Main.M4,
                io_fbFFHWO:=				GVL_PMPS.fbFastFaultOutput1,
                fbArbiter:=					GVL_PMPS.fbArbiter,
                bExecuteMotion:=			bExecuteMotion,
                bMoveOk:=					bMoveOk
);

END_PROGRAM

// ---- Spectometer Arm POUs/PRG_OPT_YG.TcPOU

PROGRAM PRG_OPT_YG
VAR
    bDebug: BOOL;
    bExecuteMotion: BOOL := TRUE;
    bMoveOk: BOOL :=TRUE;
    {attribute 'pytmc' := 'pv: QRIX:OPT'}
    fbYGMotion: FB_3AxesJack;

    bInit: BOOL :=TRUE;

    tonDelayUpdate: TON;
END_VAR


IF bInit THEN
    bInit := FALSE;

    Main.M7.nBrakeMode := ENUM_StageBrakeMode.NO_BRAKE;
    Main.M7.bHardwareEnable := TRUE;
    Main.M7.bPowerSelf := TRUE;

    Main.M8.nBrakeMode := ENUM_StageBrakeMode.NO_BRAKE;
    Main.M8.bHardwareEnable := TRUE;
    Main.M8.bPowerSelf := TRUE;

    Main.M9.nBrakeMode := ENUM_StageBrakeMode.NO_BRAKE;
    Main.M9.bHardwareEnable := TRUE;
    Main.M9.bPowerSelf := TRUE;

    Main.M7.nEnableMode := ENUM_StageEnableMode.DURING_MOTION ;
    Main.M8.nEnableMode := ENUM_StageEnableMode.DURING_MOTION ;
    Main.M9.nEnableMode := ENUM_StageEnableMode.DURING_MOTION ;
END_IF

fbYGMotion(
    bMoveOk			:= bMoveOk,
    stJack1Axis		:= Main.M9,
    stJack2Axis		:= Main.M7,
    stJack3Axis		:= Main.M8,
    rDistanceX        := 0.24,
    rDistanceZ        := 0.88,
    bJack3DoesPitch   :=  FALSE,
    rLimitPositionMax :=  8.0,
    rLimitPositionMin := -8.0,
    rLimitPitchMin    := -18,
    rLimitPitchMax    :=  18,
    rLimitRollMin     := -18,
    rLimitRollMax     :=  18,
    fMaxVelocity      :=  0.1,
);

END_PROGRAM

// ---- Spectometer Arm POUs/PRG_OPT_XPM.TcPOU

PROGRAM PRG_OPT_XPM
VAR
    bInit: BOOL :=TRUE;
    {attribute 'pytmc' := 'pv: QRIX:PM'}
    fb2AxesXPM: FB_2AxesTrans;
    bExecuteMotionXPM: BOOL :=TRUE;
    bMoveOkXPM: BOOL :=TRUE;
END_VAR

VAR CONSTANT
    rDistance	:REAL	:=	0.4;
END_VAR


IF bINIT THEN

    Main.M12.nBrakeMode := ENUM_StageBrakeMode.NO_BRAKE;
    Main.M12.bHardwareEnable := TRUE;
    Main.M12.bPowerSelf := TRUE;
    Main.M12.fVelocity := 0.1;

    Main.M13.nBrakeMode := ENUM_StageBrakeMode.NO_BRAKE;
    Main.M13.bHardwareEnable := TRUE;
    Main.M13.bPowerSelf := TRUE;
    Main.M13.fVelocity := 0.1;

    Main.M12.nEnableMode := ENUM_StageEnableMode.DURING_MOTION ;
    Main.M13.nEnableMode := ENUM_StageEnableMode.DURING_MOTION ;

    bINIT := FALSE;
END_IF;

fb2AxesXPM(	i_DevName		:=	'OPT_XPM',
            stFirstAxis		:=	Main.M12,
            stSecondAxis	:=	Main.M13,
            bExecuteMotion	:=	bExecuteMotionXPM,
            io_fbFFHWO		:=	GVL_PMPS.fbFastFaultOutput1,
            fbArbiter		:=	GVL_PMPS.fbArbiter,
            rDistance		:=	rDistance,//actually 0.48m?? //0.4, // 0.4m
            bMoveOk			:= bMoveOkXPM
);

END_PROGRAM

// ---- Devices/FB_2AxesTrans.TcPOU

FUNCTION_BLOCK FB_2AxesTrans
VAR_IN_OUT
    stFirstAxis: ST_MotionStage;
    stSecondAxis: ST_MotionStage;
    bExecuteMotion:BOOL ;
    io_fbFFHWO    :    FB_HardwareFFOutput;
    fbArbiter: FB_Arbiter();
END_VAR
VAR_INPUT

    {attribute 'pytmc' := '
    pv: PMPS_OK;
    io: i;
    field: ZNAM False
    field: ONAM True
    '}
    bMoveOk:BOOL;

    (*Offsets*)
    rEncoderOffsetFirst: REAL;
    rEncoderOffsetSecound: REAL;

    (*Distance between 1st stage and 2nd stage*)
    rDistance: REAL := 0.48;

    i_DevName : STRING; //device name for FFO and PMPS diagnostics

    bHome:BOOL:=FALSE;
END_VAR
VAR
    fbFirstStage: FB_MotionStage;
    fbSecondStage: FB_MotionStage;
    fPosFirstStage: LREAL;
    fPosSecondStage: LREAL;

    (*Motion Parameters*)
    fSmallDelta: LREAL := 0.01;
    fBigDelta: LREAL := 10;
    fMaxVelocity: LREAL := 0.03;
    fHighAccel: LREAL := 0.8;
    fLowAccel: LREAL := 0.1;

    stFirst: ST_PositionState;
    stSecond: ST_PositionState;

    {attribute 'pytmc' := 'pv: FIRST'}
    fbFirst: FB_StatePTPMove;
    {attribute 'pytmc' := 'pv: SECOND'}
    fbSecond: FB_StatePTPMove;

    (*EPICS pvs*)
    {attribute 'pytmc' := '
    pv: X_REQ;
    io: io;
    '}
    rReqPosition : REAL;
    {attribute 'pytmc' := '
    pv: PITCH_REQ;
    io: io;
    '}
    rReqAngle : REAL;


    {attribute 'pytmc' := '
    pv: X;
    io: i;
    '}
    rActPosition : REAL;

    {attribute 'pytmc' := '
    pv: PITCH;
    io: i;
    '}
    rActAngle : REAL;



     {attribute 'pytmc' := '
    pv: HOME_READY;
    io: i;
    field: ZNAM False
    field: ONAM True
    '}
    bHomeReady:BOOL:=FALSE;


    //Local variables
    bInit: BOOL :=true;
    rTrig_Block: R_TRIG;
    rTrig_Open: R_TRIG;
    rTrig_Close: R_TRIG;

    //old values
    rOldReqPosition : REAL;
    rOldReqAngle: REAL;

    bExecuteMotionX: BOOL;


    fPosBlock: LREAL;
    fPosClose: LREAL;
    fPosOpen: LREAL;

    stSetPositionOptions: ST_SetPositionOptions;
    fbSetPosition_Pos: MC_SetPosition;
    fbSetPosition_Angle: MC_SetPosition;

    // For logging
    fbLogger : FB_LogMessage := (eSubsystem:=E_SubSystem.MOTION);
    tErrorPresent : R_TRIG;
    tAction : R_TRIG;
    tOverrideActivated : R_TRIG;

    FFO    :    FB_FastFault :=(
        i_DevName := 'OPT_XPM_Translation',
        i_Desc := 'Fault occurs when center is greated than that requested',
        i_TypeCode := 16#1010);


    bTest: BOOL;

    AptArrayStatus AT %Q* : ST_PMPS_Aperture_IO;
    AptArrayReq AT %I* : ST_PMPS_Aperture_IO;
END_VAR


// Initialize
ACT_init();

// Instantiate Function block for all the blades
ACT_Motion();

//SET and GET the requested and Actual values
ACT_CalculatePositions();

ACTION ACT_CalculatePositions:

//check if requested center or gap has changed
//check that the requested values are within acceptable motion range
IF (rOldReqPosition <> rReqPosition) THEN
        rOldReqPosition := rReqPosition;
        bExecuteMotionX := TRUE;
        fbLogger(sMsg:='Requested new Position.', eSevr:=TcEventSeverity.Verbose);
END_IF

IF (rOldReqAngle <> rReqAngle) THEN
    rOldReqAngle := rReqAngle;
    bExecuteMotionX := TRUE;
    fbLogger(sMsg:='Requested new Angle', eSevr:=TcEventSeverity.Verbose);
END_IF


//Calculate requested target positions from requested gap and center
fPosFirstStage		:= rReqPosition - rDistance / 2 * rReqAngle + rEncoderOffsetFirst;
fPosSecondStage		:= rReqPosition + rDistance / 2 * rReqAngle + rEncoderOffsetSecound;



//Calculate actual gap and center from actual stages positions
rActPosition	:= LREAL_TO_REAL( ((stFirstAxis.stAxisStatus.fActPosition - rEncoderOffsetFirst) + (stSecondAxis.stAxisStatus.fActPosition - rEncoderOffsetSecound)) / 2 );
rActAngle		:= LREAL_TO_REAL( ((stSecondAxis.stAxisStatus.fActPosition - rEncoderOffsetSecound) - (stFirstAxis.stAxisStatus.fActPosition - rEncoderOffsetFirst)) / rDistance );
END_ACTION

ACTION ACT_Init:

//  init the motion stages parameters
IF ( bInit) THEN
    stFirstAxis.bHardwareEnable := TRUE;
    stSecondAxis.bHardwareEnable := TRUE;
    stFirstAxis.bPowerSelf :=TRUE;
    stSecondAxis.bPowerSelf :=TRUE;
    stFirstAxis.nBrakeMode := ENUM_StageBrakeMode.NO_BRAKE;
    stSecondAxis.nBrakeMode := ENUM_StageBrakeMode.NO_BRAKE;
    FFO.i_DevName := i_DevName;
END_IF
END_ACTION

ACTION ACT_Motion:

// Instantiate Function block for all the blades
fbFirstStage(stMotionStage:=stFirstAxis);
fbSecondStage(stMotionStage:=stSecondAxis);



// PTP Motion for each blade
stFirst.sName := 'First';
stFirst.fPosition := fPosFirstStage;
stFirst.fDelta := fSmallDelta;
stFirst.fVelocity := fMaxVelocity;
stFirst.fAccel := fHighAccel;
stFirst.fDecel := fHighAccel;

stSecond.sName := 'Second';
stSecond.fPosition := fPosSecondStage;
stSecond.fDelta := fSmallDelta;
stSecond.fVelocity := fMaxVelocity;
stSecond.fAccel := fHighAccel;
stSecond.fDecel := fHighAccel;



IF (bExecuteMotionX) THEN
    fbFirst.bExecute := fbSecond.bExecute := bExecuteMotionX;
    bExecuteMotionX:= FALSE;
END_IF


fbFirst(
    stPositionState:=stFirst,
    bMoveOk:=bMoveOk,
    stMotionStage:=stFirstAxis);

fbSecond(
    stPositionState:=stSecond,
    bMoveOk:=bMoveOk,
    stMotionStage:=stSecondAxis);
END_ACTION

END_FUNCTION_BLOCK

// ---- Spectometer Arm POUs/PRG_OPT.TcPOU

PROGRAM PRG_OPT
VAR
    bInit: BOOL := TRUE;
    fbMotionRxG: FB_MotionStage;
    fbMotionXG: FB_MotionStage;
    fbMotionRzPM: FB_MotionStage;
END_VAR


IF bInit THEN

    Main.M10.nBrakeMode := ENUM_StageBrakeMode.NO_BRAKE;
    Main.M10.bHardwareEnable := TRUE;
    Main.M10.bPowerSelf := TRUE;
    Main.M10.fVelocity := 0.1;

    Main.M11.nBrakeMode := ENUM_StageBrakeMode.NO_BRAKE;
    Main.M11.bHardwareEnable := TRUE;
    Main.M11.bPowerSelf := TRUE;
    Main.M11.fVelocity := 0.1;

    Main.M14.nBrakeMode := ENUM_StageBrakeMode.NO_BRAKE;
    Main.M14.bHardwareEnable := TRUE;
    Main.M14.bPowerSelf := TRUE;
    Main.M14.fVelocity := 0.1;

    Main.M10.nEnableMode := ENUM_StageEnableMode.DURING_MOTION ;
    Main.M11.nEnableMode := ENUM_StageEnableMode.DURING_MOTION ;
    Main.M14.nEnableMode := ENUM_StageEnableMode.DURING_MOTION ;

    bInit := FALSE;
END_IF;


fbMotionRxG(stMotionStage:= Main.M10);
fbMotionXG(stMotionStage:= Main.M11);
fbMotionRzPM(stMotionStage:= Main.M14);

END_PROGRAM

// ---- Spectometer Arm POUs/PRG_Sensor.TcPOU

PROGRAM PRG_Sensor
VAR
    bInit : bool :=TRUE;

    {attribute 'TcLinkTo' := 'TIIB[Rack#2D LinearGaugeAmp (SC-HG1-ETC)]^Process Data(Out) RxPDO-Map^Head Value Mode'}
    bSensorHeadValueMode AT %Q* : bool;

    {attribute 'TcLinkTo' := 'TIIB[Rack#2D LinearGaugeAmp (SC-HG1-ETC)]^Process Data(Out) RxPDO-Map^Normal Value Mode'}
    bSensorHeadNormalValueMode AT %Q* : bool;

    bResetSensorMode AT %I* : bool;

    uintTest AT %Q*: UINT;

END_VAR


If bInit Then
    bSensorHeadNormalValueMode := True;
    bInit := False;
End_If;

If(bResetSensorMode = True) Then
    bResetSensorMode := False;
    bSensorHeadValueMode := False;
    bSensorHeadNormalValueMode := False;
    bInit := True;
End_If;


GVL_Sensor.stYDF1.sName			:= 'YDF1 Panasonic HG-S';
GVL_Sensor.stYDF1.sEGU			:= 'mm';
GVL_Sensor.stYDF1.fCntsInEGU	:= 10000;
GVL_Sensor.nYDF1                := DINT_TO_UDINT(GVL_Sensor.stYDF1.iRawCnts + 10000);

GVL_Sensor.stYDF2.sName			:= 'YDF2 Panasonic HG-S';
GVL_Sensor.stYDF2.sEGU			:= 'mm';
GVL_Sensor.stYDF2.fCntsInEGU	:= 10000;
GVL_Sensor.nYDF2                := DINT_TO_UDINT(GVL_Sensor.stYDF2.iRawCnts + 10000);

GVL_Sensor.stYDF3.sName			:= 'YDF3 Panasonic HG-S';
GVL_Sensor.stYDF3.sEGU			:= 'mm';
GVL_Sensor.stYDF3.fCntsInEGU	:= 10000;
GVL_Sensor.nYDF3                := DINT_TO_UDINT(GVL_Sensor.stYDF3.iRawCnts + 10000);

GVL_Sensor.stHDF.sName			:= 'HDF Panasonic HG-S';
GVL_Sensor.stHDF.sEGU			:= 'mm';
GVL_Sensor.stHDF.fCntsInEGU		:= 10000;

GVL_Sensor.stGraniteP.sName		:= 'Granite Pitch';
GVL_Sensor.stGraniteP.sEGU		:= 'mrad';
GVL_Sensor.stGraniteP.fCntsInEGU:= 3276.7; // 1V = 1mrad in Low gain mode
GVL_Sensor.stGraniteP.iOffset   := -1005;
GVL_Sensor.stGraniteR.sName		:= 'Granite Roll';
GVL_Sensor.stGraniteR.sEGU		:= 'mrad';
GVL_Sensor.stGraniteR.fCntsInEGU:= 3276.7;
GVL_Sensor.stGraniteR.iOffset   := 3326;

GVL_Sensor.stFrameP.sName		:= 'Det. Frame Pitch';
GVL_Sensor.stFrameP.sEGU		:= 'mrad';
GVL_Sensor.stFrameP.fCntsInEGU	:= 3276.7;
GVL_Sensor.stFrameR.sName		:= 'Det. Frame Roll';
GVL_Sensor.stFrameR.sEGU		:= 'mrad';
GVL_Sensor.stFrameR.fCntsInEGU	:= 3276.7;

GVL_Sensor.stPS1.sName			:= 'PS1';
GVL_Sensor.stPS1.sEGU			:= 'MPa';
GVL_Sensor.stPS1.fCntsInEGU		:= 13106.8;	// 0.25MPa/V
GVL_Sensor.stPS1.iOffset		:= 3277;	// 0MPa@1V  P=0.25(V-V0), V0 = 1.0

GVL_Sensor.stPS2.sName			:= 'PS2';
GVL_Sensor.stPS2.sEGU			:= 'MPa';
GVL_Sensor.stPS2.fCntsInEGU		:= 13106.8;	// 0.25MPa/V
GVL_Sensor.stPS2.iOffset		:= 3277;	// 0MPa@1V  P=0.25(V-V0), V0 = 1.0

GVL_Sensor.stPS3.sName			:= 'PS3';
GVL_Sensor.stPS3.sEGU			:= 'MPa';
GVL_Sensor.stPS3.fCntsInEGU		:= 13106.8;	// 0.25MPa/V
GVL_Sensor.stPS3.iOffset		:= 3277;	// 0MPa@1V  P=0.25(V-V0), V0 = 1.0

GVL_Sensor.stYDF1.fValue		:= DINT_TO_REAL(GVL_Sensor.stYDF1.iRawCnts - GVL_Sensor.stYDF1.iOffset) / GVL_Sensor.stYDF1.fCntsInEGU;
GVL_Sensor.stYDF2.fValue		:= DINT_TO_REAL(GVL_Sensor.stYDF2.iRawCnts - GVL_Sensor.stYDF2.iOffset) / GVL_Sensor.stYDF2.fCntsInEGU;
GVL_Sensor.stYDF3.fValue		:= DINT_TO_REAL(GVL_Sensor.stYDF3.iRawCnts - GVL_Sensor.stYDF3.iOffset) / GVL_Sensor.stYDF3.fCntsInEGU;
GVL_Sensor.stHDF.fValue			:= DINT_TO_REAL(GVL_Sensor.stHDF.iRawCnts  - GVL_Sensor.stHDF.iOffset)  / GVL_Sensor.stHDF.fCntsInEGU;
GVL_Sensor.stGraniteP.fValue	:= -1 * INT_TO_REAL(GVL_Sensor.stGraniteP.iRawCnts - GVL_Sensor.stGraniteP.iOffset) / GVL_Sensor.stGraniteP.fCntsInEGU;
GVL_Sensor.stGraniteR.fValue	:= INT_TO_REAL(GVL_Sensor.stGraniteR.iRawCnts - GVL_Sensor.stGraniteR.iOffset) / GVL_Sensor.stGraniteR.fCntsInEGU;
GVL_Sensor.stFrameP.fValue		:= INT_TO_REAL(GVL_Sensor.stFrameP.iRawCnts - GVL_Sensor.stFrameP.iOffset) / GVL_Sensor.stFrameP.fCntsInEGU;
GVL_Sensor.stFrameR.fValue		:= -1 * INT_TO_REAL(GVL_Sensor.stFrameR.iRawCnts - GVL_Sensor.stFrameR.iOffset) / GVL_Sensor.stFrameR.fCntsInEGU;

GVL_Sensor.stPS1.fValue			:= INT_TO_REAL(GVL_Sensor.stPS1.iRawCnts - GVL_Sensor.stPS1.iOffset) / GVL_Sensor.stPS1.fCntsInEGU;
GVL_Sensor.stPS2.fValue			:= INT_TO_REAL(GVL_Sensor.stPS2.iRawCnts - GVL_Sensor.stPS2.iOffset) / GVL_Sensor.stPS2.fCntsInEGU;
GVL_Sensor.stPS3.fValue			:= INT_TO_REAL(GVL_Sensor.stPS3.iRawCnts - GVL_Sensor.stPS3.iOffset) / GVL_Sensor.stPS3.fCntsInEGU;


//uintTest:= REAL_TO_UINT(GVL_Sensor.stYDF1.fValue);

END_PROGRAM

// ---- POUs/PRG_Cryo.TcPOU

PROGRAM PRG_Cryo
VAR
    nCryoRotOutEncoderCounts AT %Q*: ULINT;
    nCryoRotEncoderOffset: ULINT;
    nDiffThetaOutEncoderCounts AT %Q*: ULINT;
    nDiffThetaEncoderOffset: ULINT;
    fb_Cryo_ROT : FB_MotionStage;
    fb_Cryo_X : FB_MotionStage;
    fb_Cryo_Y : FB_MotionStage;
    fb_Cryo_Z : FB_MotionStage;

    fbEPSCryoXBackward : FB_EPS;
    fbEPSCryoXForward  : FB_EPS;
    fbEPSCryoYBackward : FB_EPS;
    fbEPSCryoYForward  : FB_EPS;
    fbEPSCryoZBackward : FB_EPS;
    fbEPSCryoZForward  : FB_EPS;
    fbEPSCryoThetaBackward : FB_EPS;
    fbEPSCryoThetaForward  : FB_EPS;

    bInit : BOOl := TRUE;

    nGantryTolerance: LINT;
    {attribute 'pytmc' := '
        pv: QRIX:CRYO:ROT:bExecuteCouple
        io: io
        field: DESC Write TRUE to couple cryo rotation axis with diffractometer theta axis.
    '}
    bCryoRotDiffThetaExecuteCouple: BOOL := FALSE;
    {attribute 'pytmc' := '
        pv: QRIX:CRYO:ROT:bExecuteDecouple
        io: io
        field: DESC Write FALSE to decouple cryo rotation axis from diffractometer theta axis.
    '}
    bCryoRotDiffThetaExecuteDecouple: BOOL := FALSE;
    {attribute 'TcLinkTo' := '.Count := TIID^Device 2 (EtherCAT)^B950-233-WALL-S-R01-DRL-02^EL5042_03_17 - Diff - Theta - 2Theta^FB Inputs Channel 1^Position'}
    stDiffThetaEnc: ST_RenishawAbsEnc;
    {attribute 'TcLinkTo' := '.Count := TIID^Device 2 (EtherCAT)^B950-233-WALL-S-R01-DRL-01^EL5042_02_16^FB Inputs Channel 2^Position'}
    stCryoRotEnc: ST_RenishawAbsEnc;

    {attribute 'pytmc' := '
        pv: QRIX:DIFF:THETACOUPLING
        io: io
        field: DESC Structure representing cryo and diffractometer theta coupling enablement coordinator.
    '}
    stCryoRotDiffThetaAutoRealignCouple: ST_AutoRealignCouple;
    fbCryoRotDiffThetaAutoRealignCouple: FB_AutoRealignCouple;

    fbCryoRotDiffThetaCoupling: FB_GantryAutoCoupling;

    {attribute 'TcLinkTo' := '.bLeaderDriveReady := TIID^Device 2 (EtherCAT)^B950-233-WALL-S-R01-DRL-02^EL7047_03_16 - Diff - Theta^STM Status^Status^Ready;
                              .bFollowDriveReady := TIID^Device 2 (EtherCAT)^B950-233-WALL-S-R01-DRL-01^EL7047_02_11^STM Status^Status^Ready
    '}
    {attribute 'pytmc' := '
        pv: QRIX:DIFFCRYO:Coord
        io: io
        field: DESC Structure representing cryo and diffractometer theta coupling enablement coordinator.
    '}
    stCryoRotDiffThetaCoordinateGantryAxisEnable: ST_CoordinateGantryAxisEnable;
    fbCryoRotDiffThetaCoordinateGantryAxisEnable: FB_CoordinateGantryAxisEnable;

    {attribute 'TcLinkTo' := '.bFollowerDriveReady := TIID^Device 2 (EtherCAT)^B950-233-WALL-S-R01-DRL-01^EL7047_02_12^STM Status^Status^Ready
    '}
    {attribute 'pytmc' := '
        pv: QRIX:CRYO:MLC:X
        io: io
        field: DESC Structure representing Cryo X multi-leader coupling.
    '}
    stCryoXMultiLeader: ST_MultiLeaderMotionCoupling;
    fbCryoXMultiLeader: FB_MultiLeaderMotionCoupling;
    {attribute 'TcLinkTo' := '.bFollowerDriveReady := TIID^Device 2 (EtherCAT)^B950-233-WALL-S-R01-DRL-01^EL7047_02_14^STM Status^Status^Ready
    '}
    {attribute 'pytmc' := '
        pv: QRIX:CRYO:MLC:Y
        io: io
        field: DESC Structure representing Cryo Y multi-leader coupling.
    '}
    stCryoYMultiLeader: ST_MultiLeaderMotionCoupling;
    fbCryoYMultiLeader: FB_MultiLeaderMotionCoupling;
    {attribute 'TcLinkTo' := '.bFollowerDriveReady := TIID^Device 2 (EtherCAT)^B950-233-WALL-S-R01-DRL-01^EL7047_02_15^STM Status^Status^Ready
    '}
    {attribute 'pytmc' := '
        pv: QRIX:CRYO:MLC:Z
        io: io
        field: DESC Structure representing Cryo Z multi-leader coupling.
    '}
    stCryoZMultiLeader: ST_MultiLeaderMotionCoupling;
    fbCryoZMultiLeader: FB_MultiLeaderMotionCoupling;

    fCryoYNeutralPosition         : LREAL;

    {attribute 'TcLinkTo' := '.nMicrostepCounter := TIID^Device 2 (EtherCAT)^B950-233-WALL-S-R01-DRL-01^EL7047_02_11^ENC Status compact^Counter value;
                              .bCounterOverflow  := TIID^Device 2 (EtherCAT)^B950-233-WALL-S-R01-DRL-01^EL7047_02_11^ENC Status compact^Status^Counter overflow;
                              .bCounterUnderflow := TIID^Device 2 (EtherCAT)^B950-233-WALL-S-R01-DRL-01^EL7047_02_11^ENC Status compact^Status^Counter underflow'}
    fbMeasureReferenceVelocityCryoROT: FB_MeasureReferenceVelocity;
    {attribute 'TcLinkTo' := '.nMicrostepCounter := TIID^Device 2 (EtherCAT)^B950-233-WALL-S-R01-DRL-01^EL7047_02_12^ENC Status compact^Counter value;
                              .bCounterOverflow  := TIID^Device 2 (EtherCAT)^B950-233-WALL-S-R01-DRL-01^EL7047_02_12^ENC Status compact^Status^Counter overflow;
                              .bCounterUnderflow := TIID^Device 2 (EtherCAT)^B950-233-WALL-S-R01-DRL-01^EL7047_02_12^ENC Status compact^Status^Counter underflow'}
    fbMeasureReferenceVelocityCryoX: FB_MeasureReferenceVelocity;
    {attribute 'TcLinkTo' := '.nMicrostepCounter := TIID^Device 2 (EtherCAT)^B950-233-WALL-S-R01-DRL-01^EL7047_02_14^ENC Status compact^Counter value;
                              .bCounterOverflow  := TIID^Device 2 (EtherCAT)^B950-233-WALL-S-R01-DRL-01^EL7047_02_14^ENC Status compact^Status^Counter overflow;
                              .bCounterUnderflow := TIID^Device 2 (EtherCAT)^B950-233-WALL-S-R01-DRL-01^EL7047_02_14^ENC Status compact^Status^Counter underflow'}
    fbMeasureReferenceVelocityCryoY: FB_MeasureReferenceVelocity;
    {attribute 'TcLinkTo' := '.nMicrostepCounter := TIID^Device 2 (EtherCAT)^B950-233-WALL-S-R01-DRL-01^EL7047_02_15^ENC Status compact^Counter value;
                              .bCounterOverflow  := TIID^Device 2 (EtherCAT)^B950-233-WALL-S-R01-DRL-01^EL7047_02_15^ENC Status compact^Status^Counter overflow;
                              .bCounterUnderflow := TIID^Device 2 (EtherCAT)^B950-233-WALL-S-R01-DRL-01^EL7047_02_15^ENC Status compact^Status^Counter underflow'}
    fbMeasureReferenceVelocityCryoZ: FB_MeasureReferenceVelocity;
END_VAR


IF bInit THEN
    bInit := FALSE;

    Main.M46.bHardwareEnable := TRUE;
    Main.M46.bPowerSelf := TRUE;
    Main.M46.nBrakeMode := ENUM_StageBrakeMode.NO_BRAKE;
    Main.M46.nEnableMode := ENUM_StageEnableMode.DURING_MOTION;
    Main.M46.fVelocity := 0.1;

    Main.M47.bHardwareEnable := TRUE;
    Main.M47.bPowerSelf := TRUE;
    Main.M47.nBrakeMode := ENUM_StageBrakeMode.NO_BRAKE;
    Main.M47.nEnableMode := ENUM_StageEnableMode.DURING_MOTION;
    Main.M47.fVelocity := 0.1;

    Main.M48.bHardwareEnable := TRUE;
    Main.M48.bPowerSelf := TRUE;
    Main.M48.nBrakeMode := ENUM_StageBrakeMode.NO_BRAKE;
    Main.M48.nEnableMode := ENUM_StageEnableMode.DURING_MOTION;
    Main.M48.fVelocity := 0.1;

    Main.M49.bHardwareEnable := TRUE;
    Main.M49.bPowerSelf := TRUE;
    Main.M49.nBrakeMode := ENUM_StageBrakeMode.NO_BRAKE;
    Main.M49.nEnableMode := ENUM_StageEnableMode.NEVER; // ENUM_StageEnableMode.DURING_MOTION;
    Main.M49.fVelocity := 0.1;
    Main.M49.bLimitBackwardEnable := TRUE;
    Main.M49.bLimitForwardEnable := TRUE;

    // Encoder count offset in order to shift the overflow point.
    nCryoRotEncoderOffset := 1073741824;
    // Encoder count offset in order to shift the overflow point.
    nDiffThetaEncoderOffset := 1073741824;
    // 0.000000083819 deg/inc => 11,930,469.225 inc/degree
    // For 1 degree tolerance, need 11930469 inc
    nGantryTolerance := 119304690000;
    stCryoRotDiffThetaCoordinateGantryAxisEnable.bEnable := TRUE;
    // Allow setting of the reference position for gantry diff limit calculation
    stDiffThetaEnc.Ref := 121223792;
    stCryoRotEnc.Ref   := 0;

    stCryoXMultiLeader.bEnable := TRUE;
    stCryoXMultiLeader.bUseDynamicLimits := TRUE;

    GVL_VAR.fCryoYNeutralPositionAtDiffY0 := 50.7;
    stCryoYMultiLeader.bEnable := TRUE;
    stCryoYMultiLeader.bUseDynamicLimits := TRUE;

    GVL_VAR.fCryoZNeutralPositionAtDiffZ0 := 4.0;
    stCryoZMultiLeader.bEnable := TRUE;
    stCryoZMultiLeader.bUseDynamicLimits := TRUE;
END_IF

ACT_CryoThetaDiffThetaCoupling();

ACT_CryoXYZCoupling();

ACT_EPS();

fb_Cryo_X(stMotionStage:=Main.M46);
fb_Cryo_Y(stMotionStage:=Main.M47);
fb_Cryo_Z(stMotionStage:=Main.M48);
fb_Cryo_ROT(stMotionStage:=Main.M49);

fbMeasureReferenceVelocityCryoX(
    stMotionStage:=Main.M46,
    nMicrostepsPerStep:=64,
    bBusy=>,
    fMeasuredReferenceVelocity=>
);
fbMeasureReferenceVelocityCryoY(
    stMotionStage:=Main.M47,
    nMicrostepsPerStep:=64,
    bBusy=>,
    fMeasuredReferenceVelocity=>
);
fbMeasureReferenceVelocityCryoZ(
    stMotionStage:=Main.M48,
    nMicrostepsPerStep:=64,
    bBusy=>,
    fMeasuredReferenceVelocity=>
);
fbMeasureReferenceVelocityCryoROT(
    stMotionStage:=Main.M49,
    nMicrostepsPerStep:=64,
    bBusy=>,
    fMeasuredReferenceVelocity=>
);

ACTION ACT_CryoThetaDiffThetaCoupling:

// Offset the raw value to ensure the rollover point is not in the path of motion.
// offset of 90 degrees negative for -90 to 270 degree range. 90 degrees because 90/360*2^32 = 1,073,741,824.
nCryoRotOutEncoderCounts   :=  stCryoRotEnc.Count + nCryoRotEncoderOffset;
nDiffThetaOutEncoderCounts :=  UDINT_TO_ULINT(ULINT_TO_UDINT(stDiffThetaEnc.Count)) + nDiffThetaEncoderOffset;

stCryoRotEnc.Count := stCryoRotEnc.Count + nCryoRotEncoderOffset;
stDiffThetaEnc.Count := UDINT_TO_ULINT(ULINT_TO_UDINT(stDiffThetaEnc.Count)) + nDiffThetaEncoderOffset;

// Cryo Rotation and Diffractometer Theta Coupling
fbCryoRotDiffThetaCoupling(
    nGantryTol 			:= nGantryTolerance,
    Master				:= Main.M34,
    MasterEnc			:= stDiffThetaEnc,
    Slave				:= Main.M49,
    SlaveEnc			:= stCryoRotEnc,
    bExecuteCouple 		:= stCryoRotDiffThetaAutoRealignCouple.bExecuteCouple,
    bExecuteDecouple 	:= stCryoRotDiffThetaAutoRealignCouple.bExecuteDecouple
);

fbCryoRotDiffThetaAutoRealignCouple(
    stMotionStageLeader:=Main.M34,
    stMotionStageFollow:=Main.M49,
    stAutoRealignCouple:=stCryoRotDiffThetaAutoRealignCouple
);

(*fbCryoRotDiffThetaCoordinateGantryAxisEnable(
    stMotionStageLeader:=Main.M34,
    stMotionStageFollow:=Main.M49,
    stCoordinateGantryAxisEnable:=stCryoRotDiffThetaCoordinateGantryAxisEnable
);*)

IF stCryoRotDiffThetaAutoRealignCouple.bCoupled THEN
    Main.M49.nEnableMode := E_StageEnableMode.NEVER;
    Main.M49.bEnable := TRUE;
ELSE
    Main.M49.nEnableMode := E_StageEnableMode.DURING_MOTION;
END_IF
END_ACTION

ACTION ACT_CryoXYZCoupling:

IF Main.M28.bBusy THEN
    fbCryoXMultiLeader(
        stMotionStageFollow := Main.M46,
        stMultiLeaderMotionCoupling := stCryoXMultiLeader,
        fTargetPos := Main.M28.Axis.NcToPlc.ActPos,
        fTargetVel := Main.M28.Axis.NcToPlc.SetVelo,
        fTargetAcc := Main.M28.Axis.NcToPlc.SetAcc,
        bError     := Main.M28.bError,
        tTimeout   := T#5s
    );
ELSE
    fbCryoXMultiLeader(
        stMotionStageFollow := Main.M46,
        stMultiLeaderMotionCoupling := stCryoXMultiLeader,
        fTargetPos := Main.M28.Axis.NcToPlc.ActPos,
        fTargetVel := 1.0,
        fTargetAcc := 10.0,
        bError     := Main.M28.bError,
        tTimeout   := T#5s
    );
END_IF
IF stCryoXMultiLeader.bEnable AND stCryoXMultiLeader.bError THEN
    Main.M28.bError := TRUE;
END_IF

fCryoYNeutralPosition := GVL_VAR.fCryoYNeutralPositionAtDiffY0 + Main.M29.Axis.NcToPlc.ActPos;

fbCryoYMultiLeader(
    stMotionStageFollow := Main.M47,
    stMultiLeaderMotionCoupling := stCryoYMultiLeader,
    fTargetPos := F_TargetCryoYPosition(
        fNeutralPosition := GVL_VAR.fCryoYNeutralPositionAtDiffY0 + Main.M29.Axis.NcToPlc.ActPos,
        fBraidDiameter   := GVL_VAR.fBraidDiameter,
        fPhiAngleDeg     := Main.M32.Axis.NcToPlc.ActPos),
    fTargetVel := 0.5,
    fTargetAcc := 5,
    bError     := Main.M29.bError OR Main.M32.bError,
    tTimeout   := T#5s
);
IF stCryoYMultiLeader.bEnable AND stCryoYMultiLeader.bError THEN
    Main.M29.bError := TRUE;
    Main.M32.bError := TRUE;
END_IF

IF Main.M30.bBusy THEN
    fbCryoZMultiLeader(
        stMotionStageFollow:=Main.M48,
        stMultiLeaderMotionCoupling:=stCryoZMultiLeader,
        fTargetPos := fCryoZNeutralPositionAtDiffZ0 + Main.M30.Axis.NcToPlc.ActPos,
        fTargetVel := Main.M30.Axis.NcToPlc.SetVelo,
        fTargetAcc := Main.M30.Axis.NcToPlc.SetAcc,
        bError     := Main.M30.bError,
        tTimeout   := T#5s
    );
ELSE
    fbCryoZMultiLeader(
        stMotionStageFollow:=Main.M48,
        stMultiLeaderMotionCoupling:=stCryoZMultiLeader,
        fTargetPos := fCryoZNeutralPositionAtDiffZ0 + Main.M30.Axis.NcToPlc.ActPos,
        fTargetVel := 1.0,
        fTargetAcc := 10.0,
        bError     := Main.M30.bError,
        tTimeout   := T#5s
    );
END_IF
IF stCryoZMultiLeader.bEnable AND stCryoZMultiLeader.bError THEN
    Main.M30.bError := TRUE;
END_IF
END_ACTION

ACTION ACT_EPS:

// Disable movement in the negative direction.
fbEPSCryoXBackward(eps:=Main.M46.stEPSBackwardEnable);
fbEPSCryoXBackward.setDescription('NEGATIVE MOTION');
fbEPSCryoXBackward.setBit(nBits := 0,
    bValue := Main.M46.Axis.NcToPlc.ActPos - Main.M28.Axis.NcToPlc.ActPos > -1.0
);

// Disable movement in positive direction.
fbEPSCryoXForward(eps:=Main.M46.stEPSForwardEnable);
fbEPSCryoXForward.setDescription('POSITIVE MOTION');
fbEPSCryoXForward.setBit(nBits:= 0,
    bValue := Main.M46.Axis.NcToPlc.ActPos - Main.M28.Axis.NcToPlc.ActPos < 1.0
);

// Disable movement in the negative direction.
fbEPSCryoYBackward(eps:=Main.M47.stEPSBackwardEnable);
fbEPSCryoYBackward.setDescription('NEGATIVE MOTION');
fbEPSCryoYBackward.setBit(nBits := 0,
    bValue := Main.M47.Axis.NcToPlc.ActPos - F_TargetCryoYPosition(
        fNeutralPosition := GVL_VAR.fCryoYNeutralPositionAtDiffY0 + Main.M29.Axis.NcToPlc.ActPos,
        fBraidDiameter   := GVL_VAR.fBraidDiameter,
        fPhiAngleDeg     := Main.M32.Axis.NcToPlc.ActPos) > -1.0
);

// Disable movement in positive direction.
fbEPSCryoYForward(eps:=Main.M47.stEPSForwardEnable);
fbEPSCryoYForward.setDescription('POSITIVE MOTION');
fbEPSCryoYForward.setBit(nBits:= 0,
    bValue := Main.M47.Axis.NcToPlc.ActPos - F_TargetCryoYPosition(
        fNeutralPosition := GVL_VAR.fCryoYNeutralPositionAtDiffY0 + Main.M29.Axis.NcToPlc.ActPos,
        fBraidDiameter   := GVL_VAR.fBraidDiameter,
        fPhiAngleDeg     := Main.M32.Axis.NcToPlc.ActPos) < 1.0
);

// Disable movement in the negative direction.
fbEPSCryoZBackward(eps:=Main.M48.stEPSBackwardEnable);
fbEPSCryoZBackward.setDescription('NEGATIVE MOTION');
fbEPSCryoZBackward.setBit(nBits := 0,
    bValue := Main.M48.Axis.NcToPlc.ActPos - (GVL_VAR.fCryoZNeutralPositionAtDiffZ0 + Main.M30.Axis.NcToPlc.ActPos) > -1.0
);

// Disable movement in positive direction.
fbEPSCryoZForward(eps:=Main.M48.stEPSForwardEnable);
fbEPSCryoZForward.setDescription('POSITIVE MOTION');
fbEPSCryoZForward.setBit(nBits:= 0,
    bValue := Main.M48.Axis.NcToPlc.ActPos - (GVL_VAR.fCryoZNeutralPositionAtDiffZ0 + Main.M30.Axis.NcToPlc.ActPos) < 1.0
);

// Disable movement in the negative direction.
fbEPSCryoThetaBackward(eps:=Main.M49.stEPSBackwardEnable);
fbEPSCryoThetaBackward.setDescription('NEGATIVE MOTION');
fbEPSCryoThetaBackward.setBit(nBits := 0,
    bValue := Main.M49.Axis.NcToPlc.ActPos - Main.M34.Axis.NcToPlc.ActPos > -1.0
);

// Disable movement in positive direction.
fbEPSCryoThetaForward(eps:=Main.M49.stEPSForwardEnable);
fbEPSCryoThetaForward.setDescription('POSITIVE MOTION');
fbEPSCryoThetaForward.setBit(nBits:= 0,
    bValue := Main.M49.Axis.NcToPlc.ActPos - Main.M34.Axis.NcToPlc.ActPos < 1.0
);
END_ACTION

END_PROGRAM

// ---- Devices/FB_AutoRealignCouple.TcPOU

FUNCTION_BLOCK FB_AutoRealignCouple
VAR_IN_OUT
    stMotionStageLeader:  ST_MotionStage;
    stMotionStageFollow:  ST_MotionStage;
    stAutoRealignCouple:  ST_AutoRealignCouple;
END_VAR
VAR
    bInit: BOOL := TRUE;
    tTimeout: TIME;
    tStateTimeout: TIME := T#1s;
    tonTimeout: TON;
    tonRecouple: TON;
END_VAR


IF bInit THEN
    bInit := FALSE;
    stAutoRealignCouple.eState := E_RealignCoupleState.STANDBY;
END_IF

stAutoRealignCouple.bCoupled := stMotionStageLeader.Axis.NcToPlc.CoupleState = 1 AND stMotionStageFollow.Axis.NcToPlc.CoupleState = 3;

CASE stAutoRealignCouple.eState OF

    E_RealignCoupleState.STANDBY:
        IF stAutoRealignCouple.bExecute THEN
            stAutoRealignCouple.bExecute := FALSE;
            stAutoRealignCouple.eState := E_RealignCoupleState.DECOUPLE_AXES;
        END_IF
        tonTimeout(IN:=FALSE);

    E_RealignCoupleState.DECOUPLE_AXES:
        // If the gantry is already coupled, the motor is not busy, and it is enabled, then decouple the axes.
        tonTimeout(IN:=TRUE,PT:=tStateTimeout);
        IF stAutoRealignCouple.bCoupled AND NOT stMotionStageFollow.bBusy AND NOT stMotionStageFollow.bError THEN
            stAutoRealignCouple.bExecuteDecouple := TRUE;
            stAutoRealignCouple.eState := E_RealignCoupleState.COMMAND_AXES_INTO_REALIGNMENT;
            tonTimeout(IN:=FALSE);
        ELSIF NOT stAutoRealignCouple.bCoupled AND NOT stMotionStageFollow.bBusy AND NOT stMotionStageFollow.bError THEN
            stAutoRealignCouple.eState := E_RealignCoupleState.COMMAND_AXES_INTO_REALIGNMENT;
            tonTimeout(IN:=FALSE);
        ELSIF stMotionStageFollow.bError THEN
            stAutoRealignCouple.eState := E_RealignCoupleState.ERROR;
            stMotionStageFollow.bError := TRUE;
            stMotionStageFollow.sCustomErrorMessage := 'Cannot autorealign axes if the follower axis is in an error state.';
        ELSIF tonTimeout.Q THEN
            stAutoRealignCouple.eState := E_RealignCoupleState.ERROR;
            stMotionStageFollow.bError := TRUE;
            stMotionStageFollow.sCustomErrorMessage := 'Failed to decouple axes before timeout.';
        END_IF

    E_RealignCoupleState.COMMAND_AXES_INTO_REALIGNMENT:
        // If the gantry is no longer coupled, the motor is not busy, and it is enabled, then reset the decouple command and
        // command the follower axis to align with the leader axis.
        tonTimeout(IN:=TRUE,PT:=tStateTimeout);
        IF NOT stAutoRealignCouple.bCoupled AND NOT stMotionStageFollow.bBusy AND NOT stMotionStageFollow.bError THEN
            stAutoRealignCouple.bExecuteDecouple := FALSE;
            stMotionStageFollow.fPosition := stMotionStageLeader.Axis.NcToPlc.ActPos;
            stMotionStageFollow.fVelocity := stAutoRealignCouple.fRealignSpeed;
            stMotionStageFollow.bMoveCmd := TRUE;
            stAutoRealignCouple.eState := E_RealignCoupleState.WAIT_FOR_MOVE_START;
            tonTimeout(IN:=FALSE);
        ELSIF stMotionStageFollow.bError THEN
            stAutoRealignCouple.eState := E_RealignCoupleState.ERROR;
            stMotionStageFollow.bError := TRUE;
            stMotionStageFollow.sCustomErrorMessage := 'Cannot autorealign axes if the follower axis is in an error state.';
        ELSIF tonTimeout.Q THEN
            stAutoRealignCouple.eState := E_RealignCoupleState.ERROR;
            stMotionStageFollow.bError := TRUE;
            stMotionStageFollow.sCustomErrorMessage := 'Failed to decouple axes before timeout.';
            tonTimeout(IN:=FALSE);
        ELSIF NOT stMotionStageFollow.bBusy AND NOT stMotionStageFollow.bError THEN
            stAutoRealignCouple.bExecuteDecouple := TRUE;
            tonTimeout(IN:=FALSE);
        END_IF

    E_RealignCoupleState.WAIT_FOR_MOVE_START:
        // Wait for the following motor to reach the busy status, then proceed.
        tonTimeout(IN:=TRUE,PT:=tStateTimeout);
        IF stMotionStageFollow.bBusy THEN
            stAutoRealignCouple.eState := E_RealignCoupleState.RECOUPLE_AXES;

            // Estimate the amount of time it should take to make the move, use a minimum time of the state timeout time.
            tTimeout := LREAL_TO_TIME(abs(stMotionStageFollow.Axis.NcToPlc.ActPos - stMotionStageLeader.Axis.NcToPlc.ActPos) / stAutoRealignCouple.fRealignSpeed * 3.0 * 1000.0);
            IF tTimeout < tStateTimeout THEN
                tTimeout := tStateTimeout;
            END_IF

            tonTimeout(IN:=FALSE);
        ELSIF tonTimeout.Q THEN
            stAutoRealignCouple.eState := E_RealignCoupleState.ERROR;
            stMotionStageFollow.bError := TRUE;
            stMotionStageFollow.sCustomErrorMessage := 'Failed to start motor move before timeout.';
        END_IF

    E_RealignCoupleState.RECOUPLE_AXES:
        // If the follower motor is no longer busy (finished or errored or stopped) then recouple the follower motor to
        // the leader motor.
        tonTimeout(IN:=TRUE,PT:=tTimeout + T#250ms);
        tonRecouple(IN:=NOT stMotionStageFollow.bBusy AND NOT stMotionStageFollow.bError,PT:=T#250ms);
        IF tonRecouple.Q THEN
            stAutoRealignCouple.bExecuteCouple := TRUE;
            stAutoRealignCouple.eState := E_RealignCoupleState.CLEANUP;
            tonRecouple(IN:=FALSE);
        ELSIF tonTimeout.Q THEN
            stAutoRealignCouple.eState := E_RealignCoupleState.ERROR;
            stMotionStageFollow.bError := TRUE;
            stMotionStageFollow.sCustomErrorMessage := 'Failed to recouple motors after move.';
            tonRecouple(IN:=FALSE);
            tonTimeout(IN:=FALSE);
        END_IF

    E_RealignCoupleState.CLEANUP:
        // If the motors are coupled again then reinitialize the bits to
        // get them ready for another realignment attempt in the future.
        IF stAutoRealignCouple.bCoupled THEN
            stAutoRealignCouple.eState := E_RealignCoupleState.STANDBY;
            stAutoRealignCouple.bExecute := FALSE;
            stAutoRealignCouple.bExecuteDecouple := FALSE;
            stAutoRealignCouple.bExecuteCouple := FALSE;
            tonTimeout(IN:=FALSE);
        ELSE
            stAutoRealignCouple.eState := E_RealignCoupleState.RECOUPLE_AXES;
        END_IF

    E_RealignCoupleState.ERROR:
        // Timeout: In case something bad happens, have the timeout timer in place to reset the bits to guarantee we do not get
        //          stuck in this recoupling and alignment sequence.
        IF stAutoRealignCouple.bCoupled OR stMotionStageFollow.bError THEN
            stAutoRealignCouple.bExecuteCouple := FALSE;
        ELSIF NOT stMotionStageFollow.bBusy THEN
            stAutoRealignCouple.bExecuteCouple := TRUE;
        END_IF
        stAutoRealignCouple.bExecute := FALSE;
        stAutoRealignCouple.bExecuteDecouple := FALSE;
        stAutoRealignCouple.eState := E_RealignCoupleState.STANDBY;
        tonTimeout(IN:=FALSE);
        tonRecouple(IN:=FALSE);
END_CASE

END_FUNCTION_BLOCK

// ---- Devices/FB_CoordinateGantryAxisEnable.TcPOU

FUNCTION_BLOCK FB_CoordinateGantryAxisEnable
VAR_IN_OUT
    stMotionStageLeader: ST_MotionStage;
    stMotionStageFollow: ST_MotionStage;
    stCoordinateGantryAxisEnable: ST_CoordinateGantryAxisEnable;
END_VAR
VAR
    bInit: BOOL := TRUE;
    rtExecuteMove: R_TRIG;
    tonTimeout: TON;
    bMovePos: BOOL;
    bMoveNeg: BOOL;
    bMovePosAndOK: BOOL;
    bMoveNegAndOK: BOOL;
END_VAR


IF bInit THEN
    bInit := FALSE;
    stCoordinateGantryAxisEnable.eState := E_GantryEnableState.STANDBY;
END_IF

CASE stCoordinateGantryAxisEnable.eState OF

    E_GantryEnableState.STANDBY:
        IF stMotionStageLeader.bExecute AND stCoordinateGantryAxisEnable.bEnable THEN
            rtExecuteMove(CLK:=FALSE);
            stMotionStageLeader.bExecute := FALSE;
            stMotionStageLeader.bEnable := TRUE;
            stMotionStageFollow.bEnable := TRUE;
            stCoordinateGantryAxisEnable.eState := E_GantryEnableState.WAIT_FOR_FULLY_ENABLED;
        ELSIF stMotionStageLeader.bExecute AND NOT stCoordinateGantryAxisEnable.bEnable THEN
            stMotionStageLeader.bExecute := FALSE;
            stMotionStageLeader.bError := TRUE;
            stMotionStageFollow.bError := TRUE;
            stMotionStageLeader.sCustomErrorMessage := 'Move Failed. The gantry is currently disabled.';
            stMotionStageFollow.sCustomErrorMessage := stMotionStageLeader.sCustomErrorMessage;
        ELSE
            stMotionStageLeader.bEnable := FALSE;
            stMotionStageFollow.bEnable := FALSE;
        END_IF
        tonTimeout(IN:=FALSE);

    E_GantryEnableState.WAIT_FOR_FULLY_ENABLED:
        // Wait until the logic confirms both motors are fully enabled
        tonTimeout(IN:=NOT stMotionStageLeader.bAllEnable OR NOT stMotionStageFollow.bAllEnable,PT:=stCoordinateGantryAxisEnable.tTimeout);

        // Check which direction we are moving, and if the directional enables will allow that move.
        bMovePos        := stMotionStageLeader.stAxisStatus.fActPosition < stMotionStageLeader.fPosition;
        bMoveNeg        := stMotionStageLeader.stAxisStatus.fActPosition > stMotionStageLeader.fPosition;
        bMovePosAndOK   := bMovePos AND stMotionStageLeader.bAllForwardEnable AND stMotionStageFollow.bAllForwardEnable;
        bMoveNegAndOK   := bMoveNeg AND stMotionStageLeader.bAllBackwardEnable AND stMotionStageFollow.bAllBackwardEnable;

